(* IEC 61131-3 sources: volt/packages/volt-lsp-iec/test-corpus/pro2193/Device/Plc Logic/Application/09 Misc/Library Manager/L_MC1P_MotionControlBasic, 598 files *)

(* ---- L_MC1P_ABC_STATE.dut ---- *)
TYPE L_MC1P_ABC_STATE :
(
	STANDBY := 0,
	STOP := 1,
	HOMING := 2,
	JOGGING := 3,
	MOVEVEL := 4,
	MOVEABS := 5,
	MOVEREL := 6,
	EXTERNAL := 7,
	ERROR := 8,
	FINISHPOSITIONING := 9
);
END_TYPE

(* ---- L_MC1P_ADDITIONALCONFIGINFO.dut ---- *)
TYPE L_MC1P_ADDITIONALCONFIGINFO :
STRUCT
	LWIDENTDRIVESWITCHOFF : LWORD := 0;
	DWREVISION : DWORD := 0;
	DWMOTORRATEDSPEED : DWORD := 3000;
	LRREFCURRENTMOTOR : LREAL := 0;
	LRREFTORQUEMOTOR : LREAL := 1;
	LRMOTORRATEDTORQUE : LREAL := 1;
	LRTORQUELIMITFACTOR : LREAL := 1;
	LRINERTIAMOTOR : LREAL := 0.01;
	DWMOTORREVOLUTION : DWORD := 1;
	DWENCODERCRC : DWORD := 0;
	XRESETRETAINENCERRORAFTERMAINSWITCH : BOOL;
	XFEEDBACKABSPOSAVAILABLE : BOOL := TRUE;
	XVFCMODE : BOOL := FALSE;
	XTACIA402ADVANCED : BOOL := FALSE;
	WMCTRLMODEDRIVE : USINT := 1;
	XDRIVELOADENCODER : BOOL := FALSE;
	DWDRIVELOADENCODERFEEDBACKCONFIG : DWORD := 0;
	DWDRIVELOADENCODERORIENTATION : DWORD := 0;
	DWDRIVELOADENCODERCRC : DWORD := 0;
	XDEVICETRANSMITTIMESVALID : BOOL;
	LRDEVICETRANSMITTIMEACTPOSMS : LREAL;
	LRDEVICETRANSMITTIMESETPOSMS : LREAL;
END_STRUCT
END_TYPE

(* ---- L_MC1P_ADDITIONALLIMITS.dut ---- *)
TYPE L_MC1P_ADDITIONALLIMITS :
(
	NOTACTIVE := 0,
	ADDITIONALPOSLIMITS := 1
);
END_TYPE

(* ---- L_MC1P_AUTOTUNINGPARA.dut ---- *)
TYPE L_MC1P_AUTOTUNINGPARA :
STRUCT
	MAXVELOCITY : LREAL;
	MAXACCELERATION : LREAL := 0;
	MAXDISTANCE : LREAL := 0;
	MOVEMENTDISTANCE : LREAL := 0;
	STATE : WORD := 0;
	COMMANDIN : USINT;
	VPNFACTOR : WORD;
	TNNFACTOR : WORD;
	VPPFACTOR : WORD;
	VPPFACTOREXT : WORD;
	WAITINGTIME : LREAL;
END_STRUCT
END_TYPE

(* ---- L_MC1P_AXIS_STATE.dut ---- *)
TYPE L_MC1P_AXIS_STATE :
(
	ERRORSTOP := 1,
	DISABLED := 2,
	STANDSTILL := 3,
	STOPPING := 4,
	DISCMOTION := 5,
	SYNCMOTION := 6,
	CONTMOTION := 7,
	HOMING := 8,
	SERVICE := 10
);
END_TYPE

(* ---- L_MC1P_AXISBASICCONTROLINSTANCEDATA.dut ---- *)
TYPE L_MC1P_AXISBASICCONTROLINSTANCEDATA :
STRUCT
	XERROR : BOOL;
	EERRORID : L_IE1P_Error;
	XFUNBUSY : BOOL;
	XFUNDONE : BOOL;
	XFUNCOMMANDABORTED : BOOL;
	EFUNSTATEACT : L_MC1P_ABC_State;
	ABCFUNID : WORD;
	WPOWID : WORD;
	XEXIT : BOOL;
	XMOVEVELEXECUTEOLD : BOOL;
	XMOVEABSEXECUTEOLD : BOOL;
	XMOVERELEXECUTEOLD : BOOL;
	XFINISHPOSITIONINGOLD : BOOL;
	XHOMEEXECUTEOLD : BOOL;
	XJOGGINGNEGOLD : BOOL;
	XJOGGINGPOSOLD : BOOL;
	XSTOPOLD : BOOL;
	XHALTOLD : BOOL;
	XABORTOLD : BOOL;
	XPOWERROROLD : BOOL;
	XDISABLESWLIMITOLD : BOOL;
	XFUNDONEOLD : BOOL;
	XRESETHOMEPOSITIONOLD : BOOL;
	XSAVEMOVEVELDONE : BOOL;
	XACYCLICAXIS : BOOL;
	XQSPAPPLDETECTED : BOOL;
	FBSTOP_EXECUTE : BOOL;
	FBHALT_EXECUTE : BOOL;
	FBABORT_EXECUTE : BOOL;
	FBMOVEABS_EXECUTE : BOOL;
	FBMOVEVEL_EXECUTE : BOOL;
	FBMOVEREL_EXECUTE : BOOL;
	FBFINISHPOSITIONING_XFINISHPOSITIONING : BOOL;
	FBFINISHPOSITIONING_XENABLE : BOOL;
	FBJOG_XJOGPOSITIVE : BOOL;
	FBJOG_XJOGNEGATIVE : BOOL;
	FBHOME_EXECUTE : BOOL;
	FBSTOP_XINUSE : BOOL;
	FBHALT_XINUSE : BOOL;
	FBABORT_XINUSE : BOOL;
	FBMOVEABS_XINUSE : BOOL;
	FBMOVEVEL_XINUSE : BOOL;
	FBMOVEREL_XINUSE : BOOL;
	FBFINISHPOSITIONING_XINUSE : BOOL;
	FBJOG_XINUSE : BOOL;
	FBHOME_XINUSE : BOOL;
	FBBASEOLD : POINTER TO L_MC1P_Template_ForAxis;
	FBSTOP_FBBASESTATUS : L_MC1P_Template_ForAxis;
	FBHALT_FBBASESTATUS : L_MC1P_Template_ForAxis;
	FBABORT_FBBASESTATUS : L_MC1P_Template_ForAxis;
	FBHOME_FBBASESTATUS : L_MC1P_Template_ForAxis;
	FBJOG_FBBASESTATUS : L_MC1P_Template_ForAxis;
	FBMOVEABS_FBBASESTATUS : L_MC1P_Template_ForAxis;
	FBMOVEVEL_FBBASESTATUS : L_MC1P_Template_ForAxis;
	FBMOVEREL_FBBASESTATUS : L_MC1P_Template_ForAxis;
	FBFINISHPOSITIONING_FBBASESTATUS : L_MC1P_Template_ForAxis;
	FBSETFASTSTOP_FBBASESTATUS : L_MC1P_Template_ForAxis;
	FBSETFASTSTOP : L_MC1P_SetFastStop_Internal;
	FBRESET_FBBASESTATUS : L_MC1P_Template_ForAxis;
	FBRESET : L_MC1P_Reset_Internal;
	FBSETOVERRIDE_FBBASESTATUS : L_MC1P_Template_ForAxis;
	FBSETOVERRIDE : L_MC1P_SetOverride_Internal;
	FBREADMOTIONSTATE_FBBASESTATUS : L_MC1P_Template_ForAxis;
	FBREADMOTIONSTATE : L_MC1P_ReadMotionState_Internal;
	FBREADAXISERROR_FBBASESTATUS : L_MC1P_Template_ForAxis;
	FBREADAXISERROR : L_MC1P_ReadAxisError_Internal;
END_STRUCT
END_TYPE

(* ---- L_MC1P_AXISEXTENSIONTYPES.dut ---- *)
TYPE L_MC1P_AXISEXTENSIONTYPES :
(
	EMPTY := 0,
	HL9400_ECAT := 1,
	HL9400_CAN := 2,
	I500_ECAT := 3,
	I500_CAN := 4,
	I700 := 5,
	I750 := 6,
	I950 := 7,
	I950ADV := 8,
	I950_DRIVE := 9,
	I950_DRIVECIA := 10,
	GENERICDRIVE := 11,
	ENCFREE := 101,
	ENCIO_BPB := 102,
	ENCIO_ECAT := 103,
	ENCI900_ECAT := 104,
	ENCI900_DRIVE := 105,
	ENCI900_DRIVECIA := 106,
	ENCI500_ECAT := 107
);
END_TYPE

(* ---- L_MC1P_AXISFUNCTION.dut ---- *)
TYPE L_MC1P_AXISFUNCTION :
(
	SIMPLEMODE := 1,
	PLI := 2,
	MOL := 3,
	POSCTRLADAPT := 4,
	SPEEDCTRLADAPT := 5,
	SPEEDCTRLLOAD := 6,
	BRAKEGRINDIN := 7,
	BRAKETEST := 8,
	BASICBRAKECTRLONLYINDRIVE := 9,
	FLEXIBLEMAPPING := 10,
	ZEROPULS2NDFEEDBACK := 11,
	FDBSTATUSBITSAVAILABLE := 12,
	AUTOTUNING := 13,
	PARSAVEINDRIVE := 14
);
END_TYPE

(* ---- L_MC1P_AXISGUID.dut ---- *)
TYPE L_MC1P_AXISGUID :
STRUCT
	ADWDATA : ARRAY [1..4] OF DWORD;
END_STRUCT
END_TYPE

(* ---- L_MC1P_AXISPROPERTIES.dut ---- *)
TYPE L_MC1P_AXISPROPERTIES :
STRUCT
	XVIRTUAL : BOOL := FALSE;
	XTPSUPPORTED : BOOL := FALSE;
	XTPWITHTIMESTAMP : BOOL := FALSE;
	SNTPMAXCHANNEL : SINT := 0;
	XSUPPORTBRAKE : BOOL := FALSE;
	XSUPPORTDCBRAKE : BOOL := FALSE;
	XCHECKCOMMUNICATIONSTATE : BOOL := TRUE;
	XDRIVEHOMINGSUPPORTED : BOOL := FALSE;
	XTACIAADVANCED : BOOL := FALSE;
	BYDELAYLIMITDRIVEOPERATIONENABLED : BYTE := 2;
	LRTRANSMITCYCLESACTPOS : LREAL;
	LRTRANSMITCYCLESSETPOS : LREAL;
	DWTPDELAYACTPOS : DWORD;
	XFORWARDECATSLAVEERROR : BOOL := FALSE;
	XFORCEACYCLICMODE : BOOL := FALSE;
	WOFFSETDRIVEPARA : WORD := 0;
END_STRUCT
END_TYPE

(* ---- L_MC1P_AXISRETAININFO.dut ---- *)
TYPE L_MC1P_AXISRETAININFO :
STRUCT
	MEMTYPE : BYTE;
	MEMVERSION : BYTE;
	MEMLENGTH : WORD;
END_STRUCT
END_TYPE

(* ---- L_MC1P_AXISRETAININFORMATION.dut ---- *)
TYPE L_MC1P_AXISRETAININFORMATION :
STRUCT
	AXISGUID : L_MC1P_AxisGUID;
	ITFRETAIN : L_MC1P_IRetainFunction;
	PDATA : POINTER TO DWORD;
	PDATAMIRROR : POINTER TO DWORD;
END_STRUCT
END_TYPE

(* ---- L_MC1P_AXISSIMIODATA.dut ---- *)
TYPE L_MC1P_AXISSIMIODATA :
STRUCT
	XSTO : BOOL;
	XDIGIN1 : BOOL;
	XDIGIN2 : BOOL;
	XSTIMULATEERROR : BOOL;
	DWERRORCODE : DWORD;
	XQSPONERROR : BOOL;
	XSTIMULATEWARNING : BOOL;
	DWWARNINGCODE : DWORD;
	ETPMODE : UINT := 0;
	LRTPDISTANCE : LREAL;
	LRTPDISTANCEINTERNAL : LREAL;
END_STRUCT
END_TYPE

(* ---- L_MC1P_AXISSIMULATIONPDODATAFROMDRIVE.dut ---- *)
TYPE L_MC1P_AXISSIMULATIONPDODATAFROMDRIVE :
STRUCT
	UICIASTATUSWORD : UINT;
	UILENZESTATUSWORD : UINT;
	SIMODEOFOPERATIONDISP : SINT;
	UIERRORCODE : UINT;
	UITEXTREFID : UINT;
	DIVELACTVALUE : DINT;
	ITORQUEACTVALUE : INT;
	DIPOSACTVALUE : DINT;
	DIFOLLOWINGERRORACTVALUE : DINT;
	IVLACTUALVEL : INT;
	UITPSTATUS : UINT;
	DITPPOS1POSVALUE : DINT;
	DITPPOS1NEGVALUE : DINT;
	DITPPOS2POSVALUE : DINT;
	DITPPOS2NEGVALUE : DINT;
	UILENZESTATUSWORD2 : UINT;
	UDIDIGITALINPUTS : UDINT;
END_STRUCT
END_TYPE

(* ---- L_MC1P_AXISSIMULATIONPDODATAFROMDRIVESCALED.dut ---- *)
TYPE L_MC1P_AXISSIMULATIONPDODATAFROMDRIVESCALED :
STRUCT
	UICIASTATUSWORD : UINT;
	UILENZESTATUSWORD : UINT;
	SIMODEOFOPERATIONDISP : SINT;
	UIERRORCODE : UINT;
	UITEXTREFID : UINT;
	LRVELACTVALUE : LREAL;
	LRTORQUEACTVALUE : LREAL;
	LRPOSACTVALUE : LREAL;
	LRFOLLOWINGERRORACTVALUE : LREAL;
	UITPSTATUS : UINT;
	LRTPPOS1POSVALUE : LREAL;
	LRTPPOS1NEGVALUE : LREAL;
	LRTPPOS2POSVALUE : LREAL;
	LRTPPOS2NEGVALUE : LREAL;
	UILENZESTATUSWORD2 : UINT;
	UDIDIGITALINPUTS : UDINT;
END_STRUCT
END_TYPE

(* ---- L_MC1P_AXISSIMULATIONPDODATATODRIVE.dut ---- *)
TYPE L_MC1P_AXISSIMULATIONPDODATATODRIVE :
STRUCT
	UICTRLWORD : UINT;
	UILENZECTRLWORD : UINT;
	SIMODEOFOPERATION : SINT;
	ITORQUEOFFSET : INT;
	DITARGETPOSITION : DINT;
	DIVELOCITYOFFSET : DINT;
	ISPDCTRL_ILOADVALUE : INT;
	ITARGETTORQUE : INT;
	DITARGETVELOCITY : DINT;
	IVLTARGETVEL : INT;
	UITPFUNCTION1 : UINT;
	UIPOSTORQUELIMIT : UINT;
	UINEGTORQUELIMIT : UINT;
	DIUPPERSPEEDLIMIT : DINT;
	DILOWERSPEEDLIMIT : DINT;
END_STRUCT
END_TYPE

(* ---- L_MC1P_AXISSIMULATIONPDODATATODRIVESCALED.dut ---- *)
TYPE L_MC1P_AXISSIMULATIONPDODATATODRIVESCALED :
STRUCT
	UICTRLWORD : UINT;
	UILENZECTRLWORD : UINT;
	SIMODEOFOPERATION : SINT;
	LRSETPOSITION : LREAL;
	LRSETVELOCITY : LREAL;
	LRSETTORQUE : LREAL;
	LRSPDCTRL_ILOADVALUE : LREAL;
	LRVLTARGETVELOCITY : LREAL;
	UITPFUNCTION1 : UINT;
	LRPOSTORQUELIMIT : LREAL;
	LRNEGTORQUELIMIT : LREAL;
	LRUPPERSPEEDLIMIT : LREAL;
	LRLOWERSPEEDLIMIT : LREAL;
END_STRUCT
END_TYPE

(* ---- L_MC1P_AXISSIMULATIONSDODATA.dut ---- *)
TYPE L_MC1P_AXISSIMULATIONSDODATA :
STRUCT
	LRRATEDMOTORTORQUE : LREAL := 0.6;
	LRRATEDMOTORSPEED : LREAL := 4050;
	LRINERTIAMOTOR : LREAL := 0.14;
	LRINERTIALOAD : LREAL := 0;
	LRMOTORRATEDCURRENT : LREAL := 1.8;
	LRMAXMOTORSPEED : LREAL := 6075;
	BYMCTRLMODE : BYTE := 1;
	LRVP_SPEEDCTRL : LREAL := 0.00045;
	LRTN_SPEEDCTRL : LREAL := 12.8;
	LRVP_POSCTRL : LREAL := 28.4;
	LRPOSCTRLOUTPUTLIMITATION : LREAL := 480000;
	UIINSABILITYVALUE : UINT;
	UIINSABILITYINDICATOR : USINT;
	USISWITCHINGFREQUENCY : USINT := 1;
	LRPOSCTRLADAPT : LREAL := 100.0;
	LRSPEEDCTRLADAPT : LREAL := 100.0;
	LRMAXTORQUE : LREAL := 250.0;
	LRSPEEDFILTERTIME : LREAL := 0.3;
	WNBRORREVOLUTION : WORD := 1;
	DWINKPERREV : DWORD := 65536;
	DWENCODERCRC : DWORD := 1234;
	DWENCODERCRCLOAD : DWORD := 4567;
	USIBRAKEMODE : USINT := 2;
	UIBRAKESRCOFSTARTINGTORQUE : UINT := 1;
	LRBRAKEDETECTEDSTARTINGTORQUE : LREAL := 0;
	LRBRAKERELEASINGTIME : LREAL := 0.1;
	LRBRAKECLOSINGTIME : LREAL := 0.1;
	USIBRAKEOVERRIDE : USINT := 0;
	LRSTARTTORQUE : LREAL;
	UIBRAKELOGICSTATE : UINT;
	UICONTROLMODECIA402ADVANCED : UINT := 0;
	LRVP_LOADPOSCTRL : LREAL := 20.0;
	SIIPOTIMEEXP : SINT;
	USIIPOTIME : USINT;
	UIQSPOPTION : UINT;
	UDIPOSITIONREACHEDWINDOW : UDINT := 1000;
	UDIQSPDECELERATION : UDINT := 2147483647;
	DWREVISIONNBR : DWORD := 16#20000;
	DWFIRSTSYNCTIME : DWORD;
	USISPEEDERRORRESPONSE : USINT;
	SSWVERSION : STRING(50) := '1.7.5.2420 (release)';
	USIDISABLEPDOS : USINT;
	USIDRIVECOMMAND_0X2825 : USINT;
	UDIMAINSWITCHINGCYCLES_0X2D81_4 : UDINT := 666;
	USIPOSSETMODE_0X2984 : USINT;
	LRVLACCDELTASPEED : LREAL := 0;
	LRVLACCDELTATIME : LREAL := 10;
	LRVLDECDELTASPEED : LREAL := 0;
	LRVLDECDELTATIME : LREAL := 0;
	BYDISABLEDEVICE : BYTE;
	LRADDSPEEDLIMITATION : LREAL := 0;
	AUIGAINCHARACTERISTIC : ARRAY [1..11] OF WORD := [10, 100, 100, 100, 1000, 100, 2000, 100, 5000, 100, 0];
END_STRUCT
END_TYPE

(* ---- L_MC1P_AXISSLOT.dut ---- *)
TYPE L_MC1P_AXISSLOT :
(
	AXISA := 16#0,
	AXISB := 16#800
);
END_TYPE

(* ---- L_MC1P_BACKLASHCONTACTSTATE.dut ---- *)
TYPE L_MC1P_BACKLASHCONTACTSTATE :
(
	NOCONTACT := 0,
	NEGATIVECONTACT := 1,
	POSITIVECONTACT := 2
);
END_TYPE

(* ---- L_MC1P_BRAKEAUTOSTATE.dut ---- *)
TYPE L_MC1P_BRAKEAUTOSTATE :
(
	AS_IDLE,
	AS_RAMPDOWN,
	AS_CLOSINGBRAKE,
	AS_INITBRAKECLOSE,
	AS_BRAKECLOSED,
	AS_RELEASINGBRAKE,
	AS_SUPERVISORMODE,
	AS_DIRECTCONTROL
);
END_TYPE

(* ---- L_MC1P_BRAKECMDBRAKEGRINDINPARA.dut ---- *)
TYPE L_MC1P_BRAKECMDBRAKEGRINDINPARA :
STRUCT
	MOTORSPEED : INT := 1000;
	RAMPTIME : INT := 1000;
	ONTIME : INT := 500;
	OFFTIME : INT := 500;
	CYCLES : WORD := 4;
	GRINDINCONTROL : BYTE;
	MODE : USINT;
	CYCLESOUT : WORD;
	STATE : WORD;
	POSLIMIT1 : LREAL;
	POSLIMIT2 : LREAL;
END_STRUCT
END_TYPE

(* ---- L_MC1P_BRAKECMDBRAKETESTPARA.dut ---- *)
TYPE L_MC1P_BRAKECMDBRAKETESTPARA :
STRUCT
	MOTORTORQUE : DINT := 0;
	RAMPTIME : INT := 1000;
	HOLDTIME : INT := 4000;
	POSTHRESHOLD : INT;
	STATE : WORD := 0;
	WBRAKETESTMODE : USINT;
END_STRUCT
END_TYPE

(* ---- L_MC1P_BRAKECTRL.dut ---- *)
TYPE L_MC1P_BRAKECTRL :
STRUCT
	XDISABLEPHIERR : BOOL;
	XBRAKEFQSP : BOOL;
	XTORQUETIMEOUT : BOOL;
	XRELEASED : BOOL;
	XOUTPUTRELEASEOLD : BOOL;
	XOBSERVE : BOOL;
	XMODULENOTOK : BOOL;
	XEXTSIGNOTOK : BOOL;
	XMODULEFEEDBACK : BOOL;
	XBRAKEOPENED : BOOL;
	XBRAKECLOSED : BOOL;
	XINVERTBRAKE : BOOL;
	XINVERTBRAKEOLD : BOOL;
	XUVDETECTEDOLD : BOOL;
	XACTSPEEDBELOWMINSPEED : BOOL;
	XBIT15 : BOOL;
END_STRUCT
END_TYPE

(* ---- L_MC1P_BRAKEERRORCODES.dut ---- *)
TYPE L_MC1P_BRAKEERRORCODES :
(
	EC_POSITIONDRIFT := 3,
	EC_POSITIONDRIFTCINH := 11,
	EC_RAMPWATCH := 4,
	EC_ERRORMODULE := 5,
	EC_ERROREXTSIGNAL := 13,
	EC_ERRORTORQUETIMEOUT := 18,
	EC_ERRORBRAKESTATEINVALID := 19,
	EC_ERRORBRAKEMODEINVALID := 20,
	EC_TORQUELIMITED := 30
);
END_TYPE

(* ---- L_MC1P_BRAKEGRINDINSTATE.dut ---- *)
TYPE L_MC1P_BRAKEGRINDINSTATE :
(
	NOTACTIVE := 0,
	INIT := 1,
	BRAKEGRINDIN := 3,
	DONE := 4,
	ERROR := 5,
	ABORTED := 6
);
END_TYPE

(* ---- L_MC1P_BRAKELOGICSTATE.dut ---- *)
TYPE L_MC1P_BRAKELOGICSTATE :
(
	OFF := 0,
	WAITON := 1,
	SELECTPRETORQUE := 10,
	LOADPRETORQUE := 11,
	OPENBRAKE := 20,
	OPERATION := 30,
	CLOSEBRAKE := 40,
	TURNOFF := 50
);
END_TYPE

(* ---- L_MC1P_BRAKEMODE.dut ---- *)
TYPE L_MC1P_BRAKEMODE :
(
	OFF := 0,
	MANUALCONTROL_PLC := 1,
	AUTOMATIC_PLC := 2
);
END_TYPE

(* ---- L_MC1P_BRAKEOUTSTATE.dut ---- *)
TYPE L_MC1P_BRAKEOUTSTATE :
STRUCT
	XBRAKECONTROLACTIVE : BOOL;
	XMODULEOPERATION : BOOL;
	XBRAKEOUTSTATE : BOOL;
	XTORQUECTRLACTIVE : BOOL;
	XBRAKECINH : BOOL;
	XERRORACTIVE : BOOL;
	XGRINDINACTIVE : BOOL;
	XTORQUETESTACTIVE : BOOL;
	XMANOPERATION : BOOL;
	XAUTOPERATION : BOOL;
	XERROREXTFEEDBACK : BOOL;
	XERRORPOSDRIFT : BOOL;
	XERRORBRAKEMODULE : BOOL;
	XINFOTIMEOUTACTIVATE : BOOL;
	XGRINDINDONE : BOOL;
	XTORQUETESTDONE : BOOL;
	XERRORTORQUECTRL : BOOL;
	XACTSPEEDBELOWMIN : BOOL;
	XERRORTORQUELIMITED : BOOL;
END_STRUCT
END_TYPE

(* ---- L_MC1P_BRAKEPARA.dut ---- *)
TYPE L_MC1P_BRAKEPARA :
STRUCT
	LRRELEASETIME : LREAL;
	LRACTIVATIONTIME : LREAL;
	DWBRAKEMODE : DWORD;
	ESELBRAKEMODE : DWORD;
	LRSAMPLEDBRAKETORQUE : LREAL;
	LREFFECTIVESTARTINGTORQUE : LREAL;
	ALRMSTARTVALUE : ARRAY [1..2] OF LREAL;
	LRBRAKERAMPTIME : LREAL;
	XBRAKEACCDEPENDING : BOOL;
	WSOURCESTARTVALUE : WORD;
END_STRUCT
END_TYPE

(* ---- L_MC1P_BRAKESTATE.dut ---- *)
TYPE L_MC1P_BRAKESTATE :
(
	EBS_DEFAULT := 0,
	EBS_BRAKECLOSED,
	EBS_BRAKEOPEN,
	EBS_BRAKESWITCHING,
	EBS_BRAKEOBSERVATION,
	EBS_BRAKEAUTO,
	EBS_BRAKEAUTOGSB,
	EBS_BRAKEAUTOSUPERVISOR,
	EBS_BRAKEMANUAL,
	EBS_BRAKEOFF,
	EBS_STATESWITCH,
	EBS_STATEOPERATION
);
END_TYPE

(* ---- L_MC1P_BRAKETESTMODE.dut ---- *)
TYPE L_MC1P_BRAKETESTMODE :
(
	NOLOADTORQUE := 0,
	LOADTORQUEIDENTIFICATION := 1
);
END_TYPE

(* ---- L_MC1P_BRAKETESTSTATE.dut ---- *)
TYPE L_MC1P_BRAKETESTSTATE :
(
	NOTACTIVE := 0,
	INIT := 1,
	TORQUEIDENTIFICATION := 2,
	BRAKETEST := 3,
	DONE := 4,
	ERROR := 5,
	ABORTED := 6
);
END_TYPE

(* ---- L_MC1P_BUFFERDATA.dut ---- *)
TYPE L_MC1P_BUFFERDATA :
STRUCT
	LRBUFFERPOSITIONPOS : LREAL;
	LRBUFFERPOSITIONNEG : LREAL;
	LRBUFFERVELPOS : LREAL;
	LRBUFFERVELNEG : LREAL;
END_STRUCT
END_TYPE

(* ---- L_MC1P_CLASSID.dut ---- *)
TYPE L_MC1P_CLASSID :
(
	AXIS_REF := (L_MC1P_Internal.cdiEnumStartValue + 2),
	AXISBASICCONTROLV2 := (L_MC1P_Internal.cdiEnumStartValue + 3)
);
END_TYPE

(* ---- L_MC1P_COMPENSATIONMODE.dut ---- *)
TYPE L_MC1P_COMPENSATIONMODE :
(
	OFF := 0,
	AUTOMATICSET := 1,
	AUTOMATICACT := 2,
	MANUALLY := 3
);
END_TYPE

(* ---- L_MC1P_CONTROLMODE.dut ---- *)
TYPE L_MC1P_CONTROLMODE :
(
	POSCTRLDRIVE := 0,
	POSCTRLPLC := 1,
	SPEEDCTRLDRIVE := 10,
	TORQUECTRLDRIVE := 20
);
END_TYPE

(* ---- L_MC1P_CONTROLMODESET.dut ---- *)
TYPE L_MC1P_CONTROLMODESET :
(
	POSCTRLDRIVE := 0,
	POSCTRLPLC := 1,
	SPEEDCTRLDRIVE := 10
);
END_TYPE

(* ---- L_MC1P_CTRLABC.dut ---- *)
TYPE L_MC1P_CTRLABC :
STRUCT
	XREGULATORON : BOOL;
	XRESETERROR : BOOL;
	XENABLEPOSITIVE : BOOL := TRUE;
	XENABLENEGATIVE : BOOL := TRUE;
	XDISABLESWLIMIT : BOOL;
	LROVERRIDE : LREAL := 1.0;
	LROVERRIDEACC : LREAL := 1.0;
	LROVERRIDEJERK : LREAL := 1.0;
	XSTOP : BOOL;
	LRSTOPDEC : LREAL := 360000;
	LRSTOPJERK : LREAL := 0;
	XJOGGINGPOS : BOOL;
	XJOGGINGNEG : BOOL;
	XCONTINUOUSUPDATE : BOOL;
	XMOVEVELEXECUTE : BOOL;
	XMOVEABSEXECUTE : BOOL;
	XMOVERELEXECUTE : BOOL;
	XHALT : BOOL;
	LRSETPOS_DIST : LREAL;
	ESETDIRECTION : MC_DIRECTION := MC_DIRECTION.mcPositiveDirection;
	XHOMEEXECUTE : BOOL;
	LRHOMEPOSITION : LREAL;
	XUSEHOMEEXTPARAMETER : BOOL;
	SCHOMEEXTPARAMETER : L_MC1P_HomeParameter;
	SCHOMEEXTTP : MC_TRIGGER_REF;
	XHOMEABSSWITCH : BOOL;
END_STRUCT
END_TYPE

(* ---- L_MC1P_DEVICECLASS.dut ---- *)
TYPE L_MC1P_DEVICECLASS :
(
	VIRTUALAXIS := 0,
	REALAXIS := 1,
	ENCODERAXIS := 2
);
END_TYPE

(* ---- L_MC1P_DIRECTION.dut ---- *)
TYPE L_MC1P_DIRECTION :
(
	BOTH := 0,
	DIRECTIONMASTER := 1
);
END_TYPE

(* ---- L_MC1P_DRIVESPECIFICCONTAINER.dut ---- *)
TYPE L_MC1P_DRIVESPECIFICCONTAINER :
UNION
	PDATA : POINTER TO BYTE;
	BASIC : POINTER TO L_MC1P_DriveSpecific_Basic;
	CIA402 : POINTER TO L_MC1P_DriveSpecific_CiA402;
	I500 : POINTER TO L_MC1P_DriveSpecific_i500;
	I700 : POINTER TO L_MC1P_DriveSpecific_i700;
	I750 : POINTER TO L_MC1P_DriveSpecific_i750;
	I950 : POINTER TO L_MC1P_DriveSpecific_i950;
	I950ADV : POINTER TO L_MC1P_DriveSpecific_i950Adv;
	I950DRIVE : POINTER TO L_MC1P_DriveSpecific_i950_Drive;
	HL9400 : POINTER TO L_MC1P_DriveSpecific_9400HL;
	ENC : POINTER TO L_MC1P_DriveSpecific_Enc;
	ENC_BPB : POINTER TO L_MC1P_DriveSpecific_Enc_Bpb;
	ENC_FREE : POINTER TO L_MC1P_DriveSpecific_Enc_Free;
	ENC_I950 : POINTER TO L_MC1P_DriveSpecific_Enc_i950;
	ENC_I500 : POINTER TO L_MC1P_DriveSpecific_Enc_i500;
	ENC_IOECAT : POINTER TO L_MC1P_DriveSpecific_Enc_IOETC;
END_UNION
END_TYPE

(* ---- L_MC1P_DRIVESTATECOLLECTION.dut ---- *)
TYPE L_MC1P_DRIVESTATECOLLECTION :
STRUCT
	BYDRIVESTATE : BYTE;
	XDRIVETESTMODEACTIVE : BOOL;
	XDRIVEQSPACTIVE : BOOL;
	XDRIVEQSPDONE : BOOL;
	XSTOACTIVE : BOOL;
	XCINHACTIVE : BOOL;
	XVOLTAGEENABLED : BOOL;
	XUSEQSPDRIVEINSTEADOFQSPAPPL : BOOL;
	XPDOINTERFACEDISABLED : BOOL;
	XPLNOTVALID : BOOL;
	XPPIACTIVE : BOOL;
	XMAGNETISATIONFINISHED : BOOL;
	XFAULTACTIVE : BOOL;
	XFAULTREACTIONACTIVE : BOOL;
	XFIRSTERRORCYCLE : BOOL;
	XWARNINGACTIVE : BOOL;
	WTEXTREFID : WORD;
	DWDRIVEERRORID : DWORD;
	XSERVICEMODEHANDLINGINDRIVEACTIVE : BOOL;
	XBRAKESTATUSBIT : BOOL;
	XSBCACTIVE : BOOL;
END_STRUCT
END_TYPE

(* ---- L_MC1P_DRIVETYPE.dut ---- *)
TYPE L_MC1P_DRIVETYPE :
(
	VIRTUAL := 0,
	HL9400 := 1,
	I700 := 2,
	ENCODER := 3,
	GENERICDRIVE := 4,
	I500 := 5,
	I900 := 6,
	I900DRIVE := 7,
	I750 := 8,
	UNIVERSAL := 10
);
END_TYPE

(* ---- L_MC1P_ENCODERTYPE.dut ---- *)
TYPE L_MC1P_ENCODERTYPE :
(
	UNKNOWN := 0,
	FREEENCODER := 1,
	BPBENCODER := 2,
	I500ECAT := 3,
	I900ENCDRIVE := 4,
	I900ECAT := 5,
	ECATENCODER := 6
);
END_TYPE

(* ---- L_MC1P_ERRORINFORMATION.dut ---- *)
TYPE L_MC1P_ERRORINFORMATION :
STRUCT
	EERRORID : L_IE1P_Error;
	XWARNING : BOOL;
	PINSTANCE : DWORD := 0;
	TTIMESTAMP : TIME;
	TRESETTIMESTAMP : TIME;
	DWEXTENDEDERRORINFO : DWORD;
	PSINSTANCENAME : POINTER TO STRING;
END_STRUCT
END_TYPE

(* ---- L_MC1P_EXECUTIONINDEX.dut ---- *)
TYPE L_MC1P_EXECUTIONINDEX :
(
	FIRST := 1,
	SECOND := 2
);
END_TYPE

(* ---- L_MC1P_GISEQUENCE_EXFAN_LIMITS.dut ---- *)
TYPE L_MC1P_GISEQUENCE_EXFAN_LIMITS :
(
	EGI_EXFAN_LIMITS_INIT,
	EGI_EXFAN_LIMITS_FIRSTRAMP,
	EGI_EXFAN_LIMITS_SECONDRAMP,
	EGI_EXFAN_LIMITS_GENERATEPULSE,
	EGI_EXFAN_LIMITS_CHECKDISTANCE,
	EGI_EXFAN_LIMITS_CALCULATEMOVETIME,
	EGI_EXFAN_LIMITS_MOVETOLIMIT
);
END_TYPE

(* ---- L_MC1P_GISEQUENCE_EXFAN_NOLIMITS.dut ---- *)
TYPE L_MC1P_GISEQUENCE_EXFAN_NOLIMITS :
(
	EGI_EXFAN_NOLIMITS_INIT,
	EGI_EXFAN_NOLIMITS_FIRSTRAMP,
	EGI_EXFAN_NOLIMITS_SECONDRAMP,
	EGI_EXFAN_NOLIMITS_GENERATEPULSE,
	EGI_EXFAN_NOLIMITS_CHECKDIRECTION
);
END_TYPE

(* ---- L_MC1P_GISEQUENCE_NOEXFAN_LIMITS.dut ---- *)
TYPE L_MC1P_GISEQUENCE_NOEXFAN_LIMITS :
(
	EGI_NOEXFAN_LIMITS_INIT,
	EGI_NOEXFAN_LIMITS_FIRSTRAMP,
	EGI_NOEXFAN_LIMITS_SECONDRAMP,
	EGI_NOEXFAN_LIMITS_GENERATEPULSE,
	EGI_NOEXFAN_LIMITS_WAITONTIME,
	EGI_NOEXFAN_LIMITS_CHECKDISTANCE,
	EGI_NOEXFAN_LIMITS_CALCULATEMOVETIME,
	EGI_NOEXFAN_LIMITS_MOVETOLIMIT
);
END_TYPE

(* ---- L_MC1P_GISEQUENCE_NOEXFAN_NOLIMITS.dut ---- *)
TYPE L_MC1P_GISEQUENCE_NOEXFAN_NOLIMITS :
(
	EGI_NOEXFAN_NOLIMITS_INIT,
	EGI_NOEXFAN_NOLIMITS_FIRSTRAMP,
	EGI_NOEXFAN_NOLIMITS_GENERATEPULSE,
	EGI_NOEXFAN_NOLIMITS_WAITONTIME,
	EGI_NOEXFAN_NOLIMITS_CHECKDIRECTION
);
END_TYPE

(* ---- L_MC1P_GRINDINMODE.dut ---- *)
TYPE L_MC1P_GRINDINMODE :
(
	CW := 1,
	CCW := 2,
	CWCCW := 3,
	CCWCW := 4
);
END_TYPE

(* ---- L_MC1P_GRINDINSEQUENCE.dut ---- *)
TYPE L_MC1P_GRINDINSEQUENCE :
(
	EGI_DEFAULT := 0,
	EGI_INIT,
	EGI_CONTROLMODE,
	EGI_RAMP1,
	EGI_RAMP2,
	EGI_RAMPDOWN,
	EGI_PULS1,
	EGI_PULS2,
	EGI_DISABLE,
	EGI_CHOOSESTEPSEQUENCE,
	EGI_CALLSTEPSEQUENCE1,
	EGI_CALLSTEPSEQUENCE2,
	EGI_CALLSTEPSEQUENCE3,
	EGI_CALLSTEPSEQUENCE4,
	EGI_CALCULATEDOWNRAMPTYPE,
	EGI_DONE
);
END_TYPE

(* ---- L_MC1P_HOMEMODE.dut ---- *)
TYPE L_MC1P_HOMEMODE :
(
	CWTORQUELIMIT := -2,
	CCWTORQUELIMIT := -1,
	SETPOSITIONDIRECT := 0,
	CCWLIMITSWITCHCWTP := 1,
	CWLIMITSWITCHCCWTP := 2,
	CWRPCCWRNTP := 3,
	CCWRPCWRNTP := 5,
	CCWLIMITSWITCH := 17,
	CWLIMITSWITCH := 18,
	CWRPCCWRN := 19,
	CCWRPCWRN := 21,
	CCWTP := 33,
	CWTP := 34,
	SETPOSITIONINANYSTATE := 97,
	SETOFFSETINANYSTATE := 98,
	RESETHOMEINFO := 99,
	DRIVEBASED := 100
);
END_TYPE

(* ---- L_MC1P_HOMEPARAMETER.dut ---- *)
TYPE L_MC1P_HOMEPARAMETER :
STRUCT
	EHOMEMODE : L_MC1P_HomeMode;
	EHOMESTOPMODE : L_MC1P_HomeStopMode;
	LRTARGETPOSITION : LREAL;
	LRVELOCITY1 : LREAL;
	LRVELOCITY2 : LREAL;
	LRACCELERATION1 : LREAL;
	LRACCELERATION2 : LREAL;
	LRJERK : LREAL;
	RTORQUELIMIT : REAL;
	RTORQUETIME : REAL;
	DWTPCONFIG : L_MC1P_HomeTPMode;
	WDRIVEHOMEMODE : WORD;
	ESTOPMODEDIRECTION : MC_DIRECTION;
	LROFFSETPOSITION : LREAL;
END_STRUCT
END_TYPE

(* ---- L_MC1P_HOMESTOPMODE.dut ---- *)
TYPE L_MC1P_HOMESTOPMODE :
(
	STOPPOSITIONING := 0,
	RELATIVEPOSITIONING := 1,
	ABSOLUTEPOSITIONING := 2
);
END_TYPE

(* ---- L_MC1P_HOMETPMODE.dut ---- *)
TYPE L_MC1P_HOMETPMODE :
(
	EXTERNALSOURCE := 0,
	TP1_POSEDGE := 1,
	TP1_NEGEDGE := 2,
	TP1_ANYEDGE := 3,
	TP1_ZEROPULSE := 4,
	TP1_ZEROPULSE2NDFDB := 5,
	TP2_POSEDGE := 11,
	TP2_NEGEDGE := 12,
	TP2_ANYEDGE := 13,
	TP2_ZEROPULSE := 14,
	TP2_ZEROPULSEFDB2ND := 15,
	TP3_POSEDGE := 21,
	TP3_NEGEDGE := 22,
	TP3_ANYEDGE := 23,
	TP3_ZEROPULSE := 24,
	TP3_ZEROPULSEFDB2ND := 25,
	TP4_POSEDGE := 31,
	TP4_NEGEDGE := 32,
	TP4_ANYEDGE := 33,
	TP4_ZEROPULSE := 34,
	TP5_ZEROPULSEFDB2ND := 35
);
END_TYPE

(* ---- L_MC1P_I900REFOFFSETHANDLING.dut ---- *)
TYPE L_MC1P_I900REFOFFSETHANDLING :
STRUCT
	DWSWITCHCYCLECOUNTER : DWORD;
	DIDRIVEREFOFFSET : DINT;
END_STRUCT
END_TYPE

(* ---- L_MC1P_INTERNALBRAKEMODE.dut ---- *)
TYPE L_MC1P_INTERNALBRAKEMODE :
(
	BM_OFF := 0,
	BM_MANINT := 11,
	BM_AUTINT := 12,
	BM_MANEXT := 1,
	BM_AUTEXT := 2,
	BM_AUTGSB := 22
);
END_TYPE

(* ---- L_MC1P_INTERPOLATIONMODE.dut ---- *)
TYPE L_MC1P_INTERPOLATIONMODE :
(
	LINEAR := 0,
	QUADRATICPOS := 1
);
END_TYPE

(* ---- L_MC1P_INTPROFILEDATA.dut ---- *)
TYPE L_MC1P_INTPROFILEDATA :
STRUCT
	PHASE1 : L_MC1P_ProfilePhaseData;
	PHASE2 : L_MC1P_ProfilePhaseData;
	PHASE3 : L_MC1P_ProfilePhaseData;
	PHASE4 : L_MC1P_ProfilePhaseData;
	PHASE5 : L_MC1P_ProfilePhaseData;
	PHASE6 : L_MC1P_ProfilePhaseData;
	PHASE7 : L_MC1P_ProfilePhaseData;
END_STRUCT
END_TYPE

(* ---- L_MC1P_INTPROFILEDATAACC.dut ---- *)
TYPE L_MC1P_INTPROFILEDATAACC :
STRUCT
	PHASE1 : L_MC1P_ProfilePhaseData;
	PHASE2 : L_MC1P_ProfilePhaseData;
	PHASE3 : L_MC1P_ProfilePhaseData;
END_STRUCT
END_TYPE

(* ---- L_MC1P_KINDOFMOTION.dut ---- *)
TYPE L_MC1P_KINDOFMOTION :
(
	NOTDEFINED := 0,
	TRANSLATORY := 1,
	ROTARY := 2
);
END_TYPE

(* ---- L_MC1P_MAPPEDELEMENT.dut ---- *)
TYPE L_MC1P_MAPPEDELEMENT :
STRUCT
	WPARAMETER : WORD;
	WSIZE : WORD;
	PBADRESS : POINTER TO BYTE;
	PADDITIONALDATA : POINTER TO BYTE;
END_STRUCT
END_TYPE

(* ---- L_MC1P_MAPPEDOBJECTS.dut ---- *)
TYPE L_MC1P_MAPPEDOBJECTS :
STRUCT
	INDEXSUBINDEX : DWORD;
	USISIZE : USINT;
	XUSEDBYAXISREF : BOOL;
	PDATA : POINTER TO BYTE;
END_STRUCT
END_TYPE

(* ---- L_MC1P_MCTRLCONTROL.dut ---- *)
TYPE L_MC1P_MCTRLCONTROL :
(
	MCSTANDARD := 0,
	MCUF := 4,
	MCFTC := 5
);
END_TYPE

(* ---- L_MC1P_MINMAXVALUE.dut ---- *)
TYPE L_MC1P_MINMAXVALUE :
STRUCT
	LRMIN : LREAL := 0;
	LRMAX : LREAL := 0;
END_STRUCT
END_TYPE

(* ---- L_MC1P_MOLSTATE.dut ---- *)
TYPE L_MC1P_MOLSTATE :
(
	IDLE := 0,
	CHECKMOLACTIVATION := 1,
	MOLCYCLIC := 2,
	ERROR := 999
);
END_TYPE

(* ---- L_MC1P_MULTIAXISINFO.dut ---- *)
TYPE L_MC1P_MULTIAXISINFO :
STRUCT
	UIDEVICESLOT : UINT;
	UIOFFSETDRIVEPARA : UINT;
	ITFSLAVEMULTIAXISMODULEHANDLER : L_IMHP_IModuleHandler;
	ITFSLAVEAXISMODULEHANDLER : L_IMHP_IModuleHandler;
END_STRUCT
END_TYPE

(* ---- L_MC1P_ORDINALTYPE.dut ---- *)
TYPE L_MC1P_ORDINALTYPE :
(
	OTNONE := 0,
	OTBOOL := 1,
	OTBYTE := 2,
	OTSINT := 3,
	OTUSINT := 4,
	OTWORD := 5,
	OTINT := 6,
	OTUINT := 7,
	OTDWORD := 8,
	OTDINT := 9,
	OTUDINT := 10,
	OTLWORD := 11,
	OTLINT := 12,
	OTULINT := 13,
	OTREAL := 14,
	OTLREAL := 15
);
END_TYPE

(* ---- L_MC1P_PARACCESS.dut ---- *)
TYPE L_MC1P_PARACCESS :
STRUCT
	AXISNAME : REFERENCE TO STRING;
	DEVICETYPE : REFERENCE TO WORD;
	AXISSTATE : REFERENCE TO WORD;
	AXISSTATUSWORD : REFERENCE TO DWORD;
	ACTIVEERRORID : REFERENCE TO WORD;
	AXISCONTROLWORD : REFERENCE TO WORD;
	AXISCONFIGURATION : REFERENCE TO DWORD;
	ACTPOSITION : REFERENCE TO LREAL;
	ACTVELOCITY : REFERENCE TO LREAL;
	ACTACCELERATION : REFERENCE TO LREAL;
	ACTTORQUE : REFERENCE TO LREAL;
	SETPOSITION : REFERENCE TO LREAL;
	SETVELOCITY : REFERENCE TO LREAL;
	SETACCELERATION : REFERENCE TO LREAL;
	SETTORQUE : REFERENCE TO LREAL;
	KINDOFMOTIONSELECTION : REFERENCE TO WORD;
	ACTIVEUNIT : REFERENCE TO WORD;
	RATIONUMERATORADD : REFERENCE TO DWORD;
	RATIODENOMINATORADD : REFERENCE TO DWORD;
	AXISMODE : REFERENCE TO WORD;
	UDITOTALMEASURINGRANGE : REFERENCE TO UDINT;
	USEASVIRTUAL : REFERENCE TO BOOL;
	TRAVERSINGRANGE : REFERENCE TO WORD;
	CYCLELENGTH : REFERENCE TO LREAL;
	FEEDCONSTANT : REFERENCE TO LREAL;
	RATIONUMERATOR : REFERENCE TO DWORD;
	RATIODENOMINATOR : REFERENCE TO DWORD;
	ORIENTATIONINV : REFERENCE TO BOOL;
	INKPERREV : REFERENCE TO DWORD;
	INERTIALOAD : REFERENCE TO LREAL;
	INERTIAMOTOR : REFERENCE TO LREAL;
	REFTORQUE : REFERENCE TO LREAL;
	DEFAULTVELOCITY : REFERENCE TO LREAL;
	DEFAULTACCELERATION : REFERENCE TO LREAL;
	DEFAULTJERK : REFERENCE TO LREAL;
	MOTORRATEDVELOCITY : REFERENCE TO LREAL;
	MAXVELOCITY : REFERENCE TO LREAL;
	MAXACCELERATION : REFERENCE TO LREAL;
	MAXJERK : REFERENCE TO LREAL;
	DECERRORSTOP : REFERENCE TO LREAL;
	JERKERRORSTOP : REFERENCE TO LREAL;
	ENABLESWLIMIT : REFERENCE TO BOOL;
	SWLIMITPOS : REFERENCE TO LREAL;
	SWLIMITNEG : REFERENCE TO LREAL;
	BEHAVEONSWLIMIT : REFERENCE TO WORD;
	ENABLEFOLLOWINGERROR : REFERENCE TO BOOL;
	MAXFOLLOWINGERRORWARNING : REFERENCE TO LREAL;
	MAXFOLLOWINGERRORERROR : REFERENCE TO LREAL;
	ACTFOLLOWINGERROR : REFERENCE TO LREAL;
	MAXFOLLOWINGERROR : REFERENCE TO LREAL;
	FOLLOWINGERRORREACTION : REFERENCE TO WORD;
	ENCODERINPUTFILTER : REFERENCE TO USINT;
	ENCODERPOSFILTERSTATE : REFERENCE TO WORD;
	ENCODERVELFILTERSTATE : REFERENCE TO WORD;
	BTWFILTERTIME : REFERENCE TO DINT;
	REDPOSQUANT : REFERENCE TO WORD;
	ENCFILTERCYCLES : REFERENCE TO WORD;
	ENCFILTERCYCLESPOS : REFERENCE TO WORD;
	COMPENSATIONMODE : REFERENCE TO WORD;
	SETVALDELAYTIME : REFERENCE TO LREAL;
	ENCODERUPDATETIME : REFERENCE TO DWORD;
	HOMING_MODE : REFERENCE TO INT;
	HOMING_STOPMODE : REFERENCE TO INT;
	HOMING_TARGETPOSITION : REFERENCE TO LREAL;
	HOMING_VELOCITY1 : REFERENCE TO LREAL;
	HOMING_VELOCITY2 : REFERENCE TO LREAL;
	HOMING_ACCELERATION1 : REFERENCE TO LREAL;
	HOMING_ACCELERATION2 : REFERENCE TO LREAL;
	HOMING_JERK : REFERENCE TO LREAL;
	HOMING_TORQUELIMIT : REFERENCE TO REAL;
	HOMING_TORQUETIME : REFERENCE TO REAL;
	HOMING_TPCONFIG : REFERENCE TO DWORD;
	HOMING_RESTOREHOMEPOSITION : REFERENCE TO BOOL;
	HOMING_RESTORETRESHOLD : REFERENCE TO LREAL;
	HOMING_DRIVEHOMEMODE : REFERENCE TO WORD;
	HOMING_HOMEPOSITION : REFERENCE TO LREAL;
	HOMING_POSSETPERMANENTLY : REFERENCE TO USINT;
	HOMIN_OFFSETPOSITION : REFERENCE TO LREAL;
	HOMING_STOPMODEDIRECTION : REFERENCE TO INT;
	CONTROLMODEDEFAULT : REFERENCE TO WORD;
	ACTCONTROLMODE : REFERENCE TO WORD;
	ENCODERNAME : REFERENCE TO STRING;
	POSCTRLGAIN : REFERENCE TO LREAL;
	POSCTRLOUTPUTLIMITATION : REFERENCE TO LREAL;
	POSCTRKOUTPUT : REFERENCE TO LREAL;
	POSCTRLADAPTVALUE : REFERENCE TO UINT;
	POSCTRLADAPTIONFROM0X2985 : REFERENCE TO USINT;
	POSCTRLADAPTACTIVEVALUE : REFERENCE TO UINT;
	SETVALUEMONITORING : REFERENCE TO BOOL;
	TIMELIMITSWITCHON : REFERENCE TO REAL;
	REAKTONMCFBERROR : REFERENCE TO BOOL;
	ENABLELOGENTRY : REFERENCE TO BOOL;
	HWLIMITERRORREACTION : REFERENCE TO USINT;
	SWLIMITERRORREACTION : REFERENCE TO USINT;
	LIMITPROFILEERRORREACTION : REFERENCE TO USINT;
	CINHERRORREACTION : REFERENCE TO USINT;
	LIMITERSTOPREACTION : REFERENCE TO USINT;
	BRAKE_MODE : REFERENCE TO DWORD;
	BRAKE_RELEASETIME : REFERENCE TO LREAL;
	BRAKE_ACTIVATIONTIME : REFERENCE TO LREAL;
	BRAKE_ACTMODE : REFERENCE TO DWORD;
	BRAKE_SAMPLEDTORQUE : REFERENCE TO LREAL;
	BRAKE_EFFECTIVETORQUE : REFERENCE TO LREAL;
	BRAKETEST_STATE : REFERENCE TO WORD;
	BRAKE_SOURCESTARTVALUE : REFERENCE TO WORD;
	BRAKE_MSTARTVALUE : REFERENCE TO LREAL;
	BRAKE_BRAKERAMPTIME : REFERENCE TO LREAL;
	BRAKE_BRAKEACCDEPENDING : REFERENCE TO BOOL;
	BRAKETEST_CMD : REFERENCE TO USINT;
	BRAKETEST_MODE : REFERENCE TO USINT;
	BRAKETEST_TORQUE : REFERENCE TO DINT;
	BRAKETEST_THRESHOLD : REFERENCE TO INT;
	BRAKETEST_RAMPTIME : REFERENCE TO INT;
	BRAKETEST_HOLDTIME : REFERENCE TO INT;
	BRAKETEST_ACTTRESHOLD : REFERENCE TO INT;
	TORQUELIMHIGH : REFERENCE TO INT;
	TORQUELIMLOW : REFERENCE TO INT;
	WINDOWTARGETREACHED : REFERENCE TO LREAL;
	WINDOWTARGETREACHEDTIME : REFERENCE TO LREAL;
	WINDOWSTANDSTILL : REFERENCE TO LREAL;
	OPTIMIZEDPROFILECALCULATIONMODE : REFERENCE TO UINT;
	MODPOSTOLERANCE : REFERENCE TO LREAL;
	RECOVERYWINDOWPOS : REFERENCE TO LREAL;
	RECOVERYWINDOWNEG : REFERENCE TO LREAL;
	SERVICEDIRECTION : REFERENCE TO WORD;
	BRAKEGRINDIN_CMD : REFERENCE TO USINT;
	BRAKEGRINDIN_MODE : REFERENCE TO USINT;
	BRAKEGRINDIN_CTRL : REFERENCE TO BYTE;
	BRAKEGRINDIN_SPEED : REFERENCE TO INT;
	BRAKEGRINDIN_RAMPTIME : REFERENCE TO INT;
	BRAKEGRINDIN_ONTIME : REFERENCE TO INT;
	BRAKEGRINDIN_OFFTIME : REFERENCE TO INT;
	BRAKEGRINDIN_CYCLES : REFERENCE TO WORD;
	BRAKEGRINDIN_CYCLESOUT : REFERENCE TO WORD;
	BRAKEGRINDIN_STATE : REFERENCE TO WORD;
	LIMITEDVELOCITY1 : REFERENCE TO LREAL;
	LIMITEDDECELERATION1 : REFERENCE TO LREAL;
	LIMITEDVELOCITY2 : REFERENCE TO LREAL;
	LIMITEDDECELERATION2 : REFERENCE TO LREAL;
	LIMITEDVELOCITY3 : REFERENCE TO LREAL;
	LIMITEDDECELERATION3 : REFERENCE TO LREAL;
	LIMITEDVELOCITY4 : REFERENCE TO LREAL;
	LIMITEDDECELERATION4 : REFERENCE TO LREAL;
	LIMITEDDISTANCE : REFERENCE TO LREAL;
	SLSOFFSETVELOCITY : REFERENCE TO LREAL;
	FOLLOWERSLS : REFERENCE TO BOOL;
	LIMITSPEEDCTRLSLS : REFERENCE TO BOOL;
	DISABLESAFETYINTERFACE : REFERENCE TO DWORD;
	REQUESTSAFETYINTERFACE : REFERENCE TO DWORD;
	SLIDISTANCE : REFERENCE TO LREAL;
	BRAKEGRINDIN_POSLIMIT1 : REFERENCE TO LREAL;
	BRAKEGRINDIN_POSLIMIT2 : REFERENCE TO LREAL;
	AUTOTUNING_CMD : REFERENCE TO USINT;
	AT_VELOCITY : REFERENCE TO LREAL;
	AT_ACCELERATION : REFERENCE TO LREAL;
	AT_DISTANCE : REFERENCE TO LREAL;
	AT_CALCULATEDDISTANCE : REFERENCE TO LREAL;
	AT_VPNFACTOR : REFERENCE TO WORD;
	AT_TNNFACTOR : REFERENCE TO WORD;
	AT_STATE : REFERENCE TO WORD;
	AT_VPPFACTOR : REFERENCE TO WORD;
	AT_VPPFACTOREXT : REFERENCE TO WORD;
	AT_WAITINGTIME : REFERENCE TO LREAL;
	JOGGINGSETVEL : REFERENCE TO LREAL;
	JOGGINGSETACC : REFERENCE TO LREAL;
	JOGGINGSETDEC : REFERENCE TO LREAL;
	JOGGINGSETJERK : REFERENCE TO LREAL;
	HALTDEC : REFERENCE TO LREAL;
	HALTJERK : REFERENCE TO LREAL;
END_STRUCT
END_TYPE

(* ---- L_MC1P_PARAMETERDATASIM.dut ---- *)
TYPE L_MC1P_PARAMETERDATASIM :
STRUCT
	WINDEX : WORD;
	BYSUBINDEX : BYTE;
	PVALUE : POINTER TO BYTE;
	BYNROFBYTE : BYTE;
	XSUPPORTED : BOOL;
	XWRITEACCESS : BOOL;
	XAXISOFFSETSUPPORTED : BOOL;
	EFIXTOLREAL : L_MC1P_ScaleFixToLREAL := L_MC1P_ScaleFixToLREAL.None;
END_STRUCT
END_TYPE

(* ---- L_MC1P_PARAMS.dut ---- *)
TYPE L_MC1P_PARAMS :
(
	AXISNAME := 2,
	DEVICETYPE := 3,
	AXISSTATE := 4,
	AXISSTATUSWORD := 5,
	ACTIVEERRORID := 6,
	AXISCONTROLWORD := 8,
	AXISCONFIGURATION := 9,
	ACTPOSITION := 10,
	ACTVELOCITY := 11,
	ACTACCELERATION := 12,
	ACTTORQUE := 13,
	SETPOSITION := 14,
	SETVELOCITY := 15,
	SETACCELERATION := 16,
	SETTORQUE := 17,
	KINDOFMOTIONSELECTION := 20,
	ACTIVEUNIT := 21,
	RATIONUMERATORADD := 25,
	RATIODENOMINATORADD := 26,
	AXISMODE := 27,
	UDITOTALMEASURINGRANGE := 28,
	USEASVIRTUAL := 29,
	TRAVERSINGRANGE := 30,
	CYCLELENGTH := 31,
	FEEDCONSTANT := 32,
	RATIONUMERATOR := 33,
	RATIODENOMINATOR := 34,
	ORIENTATIONINV := 35,
	INKPERREV := 36,
	INERTIALOAD := 37,
	INERTIAMOTOR := 38,
	REFTORQUE := 39,
	DEFAULTVELOCITY := 40,
	DEFAULTACCELERATION := 41,
	DEFAULTJERK := 43,
	MOTORRATEDVELOCITY := 44,
	MAXVELOCITY := 45,
	MAXACCELERATION := 46,
	MAXJERK := 47,
	DECERRORSTOP := 48,
	JERKERRORSTOP := 49,
	ENABLESWLIMIT := 50,
	SWLIMITPOS := 51,
	SWLIMITNEG := 52,
	BEHAVEONSWLIMIT := 53,
	ENABLEFOLLOWINGERROR := 54,
	MAXFOLLOWINGERRORWARNING := 55,
	MAXFOLLOWINGERRORERROR := 56,
	ACTFOLLOWINGERROR := 57,
	MAXFOLLOWINGERROR := 58,
	FOLLOWINGERRORREACTION := 59,
	ENCODERINPUTFILTER := 60,
	ENCODERPOSFILTERSTATE := 61,
	ENCODERVELFILTERSTATE := 62,
	BTWFILTERTIME := 63,
	REDPOSQUANT := 64,
	ENCFILTERCYCLES := 65,
	ENCFILTERCYCLESPOS := 66,
	COMPENSATIONMODE := 67,
	SETVALDELAYTIME := 68,
	ENCODERUPDATETIME := 69,
	HOMING_MODE := 70,
	HOMING_STOPMODE := 71,
	HOMING_TARGETPOSITION := 72,
	HOMING_VELOCITY1 := 73,
	HOMING_VELOCITY2 := 74,
	HOMING_ACCELERATION1 := 75,
	HOMING_ACCELERATION2 := 76,
	HOMING_JERK := 77,
	HOMING_TORQUELIMIT := 78,
	HOMING_TORQUETIME := 79,
	HOMING_TPCONFIG := 80,
	HOMING_RESTOREHOMEPOSITION := 81,
	HOMING_RESTORETRESHOLD := 82,
	HOMING_DRIVEHOMEMODE := 83,
	HOMING_HOMEPOSITION := 84,
	HOMING_POSSETPERMANENTLY := 85,
	HOMIN_OFFSETPOSITION := 86,
	HOMING_STOPMODEDIRECTION := 87,
	CONTROLMODEDEFAULT := 90,
	ACTCONTROLMODE := 91,
	ENCODERNAME := 92,
	POSCTRLGAIN := 93,
	POSCTRLOUTPUTLIMITATION := 94,
	POSCTRKOUTPUT := 95,
	POSCTRLADAPTVALUE := 96,
	POSCTRLADAPTIONFROM0X2985 := 97,
	POSCTRLADAPTACTIVEVALUE := 98,
	SETVALUEMONITORING := 100,
	TIMELIMITSWITCHON := 101,
	REAKTONMCFBERROR := 102,
	ENABLELOGENTRY := 103,
	HWLIMITERRORREACTION := 104,
	SWLIMITERRORREACTION := 105,
	LIMITPROFILEERRORREACTION := 106,
	CINHERRORREACTION := 107,
	LIMITERSTOPREACTION := 108,
	BRAKE_MODE := 110,
	BRAKE_RELEASETIME := 111,
	BRAKE_ACTIVATIONTIME := 112,
	BRAKE_ACTMODE := 113,
	BRAKE_SAMPLEDTORQUE := 114,
	BRAKE_EFFECTIVETORQUE := 115,
	BRAKETEST_STATE := 116,
	BRAKE_SOURCESTARTVALUE := 117,
	BRAKE_MSTARTVALUE := 118,
	BRAKE_BRAKERAMPTIME := 119,
	BRAKE_BRAKEACCDEPENDING := 120,
	BRAKETEST_CMD := 121,
	BRAKETEST_MODE := 122,
	BRAKETEST_TORQUE := 123,
	BRAKETEST_THRESHOLD := 124,
	BRAKETEST_RAMPTIME := 125,
	BRAKETEST_HOLDTIME := 126,
	BRAKETEST_ACTTRESHOLD := 127,
	TORQUELIMHIGH := 128,
	TORQUELIMLOW := 129,
	WINDOWTARGETREACHED := 130,
	WINDOWTARGETREACHEDTIME := 131,
	WINDOWSTANDSTILL := 132,
	OPTIMIZEDPROFILECALCULATIONMODE := 134,
	MODPOSTOLERANCE := 135,
	RECOVERYWINDOWPOS := 136,
	RECOVERYWINDOWNEG := 137,
	SERVICEDIRECTION := 139,
	BRAKEGRINDIN_CMD := 140,
	BRAKEGRINDIN_MODE := 141,
	BRAKEGRINDIN_CTRL := 142,
	BRAKEGRINDIN_SPEED := 143,
	BRAKEGRINDIN_RAMPTIME := 144,
	BRAKEGRINDIN_ONTIME := 145,
	BRAKEGRINDIN_OFFTIME := 146,
	BRAKEGRINDIN_CYCLES := 147,
	BRAKEGRINDIN_CYCLESOUT := 148,
	BRAKEGRINDIN_STATE := 149,
	LIMITEDVELOCITY1 := 150,
	LIMITEDDECELERATION1 := 151,
	LIMITEDVELOCITY2 := 152,
	LIMITEDDECELERATION2 := 153,
	LIMITEDVELOCITY3 := 154,
	LIMITEDDECELERATION3 := 155,
	LIMITEDVELOCITY4 := 156,
	LIMITEDDECELERATION4 := 157,
	LIMITEDDISTANCE := 158,
	SLSOFFSETVELOCITY := 159,
	FOLLOWERSLS := 160,
	LIMITSPEEDCTRLSLS := 161,
	DISABLESAFETYINTERFACE := 162,
	REQUESTSAFETYINTERFACE := 163,
	SLIDISTANCE := 164,
	BRAKEGRINDIN_POSLIMIT1 := 168,
	BRAKEGRINDIN_POSLIMIT2 := 169,
	AUTOTUNING_CMD := 170,
	AT_VELOCITY := 171,
	AT_ACCELERATION := 172,
	AT_DISTANCE := 173,
	AT_CALCULATEDDISTANCE := 174,
	AT_VPNFACTOR := 175,
	AT_TNNFACTOR := 176,
	AT_STATE := 177,
	AT_VPPFACTOR := 178,
	AT_VPPFACTOREXT := 179,
	AT_WAITINGTIME := 180,
	JOGGINGSETVEL := 181,
	JOGGINGSETACC := 182,
	JOGGINGSETDEC := 183,
	JOGGINGSETJERK := 184,
	HALTDEC := 186,
	HALTJERK := 187
);
END_TYPE

(* ---- L_MC1P_PARGENERALMECHANIC.dut ---- *)
TYPE L_MC1P_PARGENERALMECHANIC :
STRUCT
	WBRAKEAVAILABLE : WORD := 0;
	LRBRAKEACTIVATIONTIME : LREAL := 0.01;
	LRCURRCTRLPT2TT_T1 : LREAL := (246.06 * 1E-06);
	LRCURRCTRLPT2TT_T2 : LREAL := (210.35 * 1E-06);
	LRCURRCTRLPT2TT_DELAY : LREAL := (103.3 * 1E-06);
END_STRUCT
END_TYPE

(* ---- L_MC1P_PARMECHANIC.dut ---- *)
TYPE L_MC1P_PARMECHANIC :
STRUCT
	LRINERTIA : LREAL := 2.99E-05;
	LRVISCOSEFACTOR : LREAL := 0.001;
	LRCOULOMBFACTOR : LREAL := 0.025;
	LRCOULOMBSLOPE : LREAL := 1;
	LREXTERNALTORQUE : LREAL;
	LRBRAKEMAXTORQUE : LREAL := 2;
	LRMECHMINPOS : LREAL := 0;
	LRMECHMAXPOS : LREAL := 0;
END_STRUCT
END_TYPE

(* ---- L_MC1P_PARMECHANIC2MS.dut ---- *)
TYPE L_MC1P_PARMECHANIC2MS :
STRUCT
	LRINERTIA2 : LREAL;
	LRD : LREAL;
	LRC : LREAL;
	LRFRICTIONRATIO : LREAL := (1.0 / 4.0);
END_STRUCT
END_TYPE

(* ---- L_MC1P_PARMECHANIC2MS_BACKLASH.dut ---- *)
TYPE L_MC1P_PARMECHANIC2MS_BACKLASH :
STRUCT
	LRBACKLASH : LREAL;
END_STRUCT
END_TYPE

(* ---- L_MC1P_PARMECHANIC3MS.dut ---- *)
TYPE L_MC1P_PARMECHANIC3MS :
STRUCT
	LRINERTIA2 : LREAL := (1.95 - 4);
	LRINERTIA3 : LREAL := 1.6E-05;
	D1 : LREAL := 2.24;
	D2 : LREAL := 0.007;
	C1 : LREAL := 2.24;
	C2 : LREAL := 0.008;
END_STRUCT
END_TYPE

(* ---- L_MC1P_PGFUTVAL.dut ---- *)
TYPE L_MC1P_PGFUTVAL :
STRUCT
	DROUTACC : LREAL;
	DROUTSPEED : LREAL;
	DROUTPOS : LREAL;
	DRCNT : LREAL;
END_STRUCT
END_TYPE

(* ---- L_MC1P_PGPHASENPARA.dut ---- *)
TYPE L_MC1P_PGPHASENPARA :
STRUCT
	DRRELTIME : LREAL;
	DRTIME : LREAL;
	DRRELPOS : LREAL;
	DRPOS : LREAL;
	DRRELSPEED : LREAL;
	DRSPEED : LREAL;
	DRRELACC : LREAL;
	DRACC : LREAL;
	DRJERKA : LREAL;
	IBPROFILENUMBER : INT;
END_STRUCT
END_TYPE

(* ---- L_MC1P_POSCTRLADAPTMODE.dut ---- *)
TYPE L_MC1P_POSCTRLADAPTMODE :
(
	MOTORANDLOAD := 0,
	MOTOR := 1,
	LOAD := 2
);
END_TYPE

(* ---- L_MC1P_POSLINT.dut ---- *)
TYPE L_MC1P_POSLINT :
UNION
	LIPOS : LINT;
	ADIPOS : ARRAY [1..2] OF DINT;
END_UNION
END_TYPE

(* ---- L_MC1P_PPISTATE.dut ---- *)
TYPE L_MC1P_PPISTATE :
(
	IDLE := 0,
	CHECKPPIACTIVATION := 1,
	PPIMONITORING := 2,
	DONE := 3,
	RESETPPIINFORMATION := 4,
	SETPPIINFORMATION := 5,
	ERROR := 999
);
END_TYPE

(* ---- L_MC1P_PRECONTROLMODE.dut ---- *)
TYPE L_MC1P_PRECONTROLMODE :
(
	AUTOMATIC := 0,
	ADDITIVEOFFSETTORQUE := 1,
	EXCLUSIVEOFFSETTORQUE := 2
);
END_TYPE

(* ---- L_MC1P_PRMDATAHEADER.dut ---- *)
TYPE L_MC1P_PRMDATAHEADER :
STRUCT
	PARAMHEADERTYPE : DWORD;
	PARAMETERDATAOFFSETFROMSTARTOF : DWORD;
	PARAMDATASIZE : DWORD;
END_STRUCT
END_TYPE

(* ---- L_MC1P_PRMFILEHEADER.dut ---- *)
TYPE L_MC1P_PRMFILEHEADER :
STRUCT
	PARSETTYPE : DWORD;
	FILEVERSION : DWORD;
	SIZETOTAL : DWORD;
	VENDOR : DWORD;
	PRODUCTCODE : DWORD;
	REVISION : DWORD;
	DATAOFFSET : DWORD;
	DATASIZE : DWORD;
	CRCCHECKSUM : DWORD;
END_STRUCT
END_TYPE

(* ---- L_MC1P_PRMPARAMETERHEADER.dut ---- *)
TYPE L_MC1P_PRMPARAMETERHEADER :
STRUCT
	SIZE : WORD;
	INDEX : WORD;
	SUBINDEX : WORD;
END_STRUCT
END_TYPE

(* ---- L_MC1P_PROFILEDATA.dut ---- *)
TYPE L_MC1P_PROFILEDATA :
STRUCT
	ALRPROFILETIME : ARRAY [0..8] OF LREAL;
	ALRPROFILEPOS : ARRAY [0..8] OF LREAL;
	ALRPROFILEVEL : ARRAY [0..8] OF LREAL;
	ALRPROFILEACC : ARRAY [0..8] OF LREAL;
	ALRPROFILEJERK : ARRAY [0..8] OF LREAL;
END_STRUCT
END_TYPE

(* ---- L_MC1P_PROFILEDATAEXTENDED.dut ---- *)
TYPE L_MC1P_PROFILEDATAEXTENDED :
STRUCT
	ALRPROFILETIME : ARRAY [0..11] OF LREAL;
	ALRPROFILEPOS : ARRAY [0..11] OF LREAL;
	ALRPROFILEVEL : ARRAY [0..11] OF LREAL;
	ALRPROFILEACC : ARRAY [0..11] OF LREAL;
	ALRPROFILEJERK : ARRAY [0..11] OF LREAL;
END_STRUCT
END_TYPE

(* ---- L_MC1P_PROFILEPARAMETER.dut ---- *)
TYPE L_MC1P_PROFILEPARAMETER :
STRUCT
	LRTARGETPOS : LREAL := 0;
	LRTARGETVEL : LREAL := 0;
	LRTARGETACC : LREAL := 0;
	LRMAXVEL : LREAL := 0;
	LRMAXACC : LREAL := 0;
	LRMAXDEC : LREAL := 0;
	LRJERKACC : LREAL := 0;
	LRJERKDEC : LREAL := 0;
END_STRUCT
END_TYPE

(* ---- L_MC1P_PROFILEPHASEDATA.dut ---- *)
TYPE L_MC1P_PROFILEPHASEDATA :
STRUCT
	T : LREAL;
	DS : LREAL;
	DV : LREAL;
	DA : LREAL;
	J : LREAL;
END_STRUCT
END_TYPE

(* ---- L_MC1P_PROFILETYPE.dut ---- *)
TYPE L_MC1P_PROFILETYPE :
(
	POLY_4TH_ORDER := 0,
	POLY_2TH_ORDER := 1,
	POLY_5TH_ORDER := 2
);
END_TYPE

(* ---- L_MC1P_QUICKSTOPOPTION.dut ---- *)
TYPE L_MC1P_QUICKSTOPOPTION :
(
	DISABLEDRIVE := 2,
	STAYINQSP := 6
);
END_TYPE

(* ---- L_MC1P_RETAINDATAENCAXIS.dut ---- *)
TYPE L_MC1P_RETAINDATAENCAXIS :
STRUCT
	XRETAININITIALIZED : BOOL;
	RETAINSTACK1 : L_MC1P_uRetainData;
	RETAINSTACK2 : L_MC1P_uRetainData;
END_STRUCT
END_TYPE

(* ---- L_MC1P_RETAINDATAI700.dut ---- *)
TYPE L_MC1P_RETAINDATAI700 :
STRUCT
	DWENCODERCRC : DWORD;
	LRBRAKESAMPLEDTORQUE : LREAL;
END_STRUCT
END_TYPE

(* ---- L_MC1P_RETAINDATAI700_V2.dut ---- *)
TYPE L_MC1P_RETAINDATAI700_V2 :
STRUCT
	DWENCODERCRC : DWORD;
	LRBRAKESAMPLEDTORQUE : LREAL;
END_STRUCT
END_TYPE

(* ---- L_MC1P_RETAINDATAI700_V3.dut ---- *)
TYPE L_MC1P_RETAINDATAI700_V3 :
STRUCT
	DWENCODERCRC : DWORD;
	LRBRAKESAMPLEDTORQUE : LREAL;
END_STRUCT
END_TYPE

(* ---- L_MC1P_RETAINDATAREALDRIVE.dut ---- *)
TYPE L_MC1P_RETAINDATAREALDRIVE :
STRUCT
	DWPROPERTIES : DWORD;
	UPOSACT : L_MC1P_PosLINT;
	DIREFOFFSETINC : DINT;
	LRACTPOS : LREAL;
	LRABSREFOFFSET : LREAL;
	LRCYCLELENGTH : LREAL;
	LRSCALEFACTOR : LREAL;
END_STRUCT
END_TYPE

(* ---- L_MC1P_RETAINDATAREALDRIVE_V2.dut ---- *)
TYPE L_MC1P_RETAINDATAREALDRIVE_V2 :
STRUCT
	DWPROPERTIES : DWORD;
	UPOSACT : L_MC1P_PosLINT;
	DIREFOFFSETINC : DINT;
	LRACTPOS : LREAL;
	LRABSREFOFFSET : LREAL;
	LRCYCLELENGTH : LREAL;
	LRSCALEFACTOR : LREAL;
	DISETPOSROUNDSLAST : DINT;
	LRLASTSETPOSITION : LREAL;
	DITARGETPOSROUNDS : DINT;
	LRLASTTARGETPOSITION : LREAL;
END_STRUCT
END_TYPE

(* ---- L_MC1P_RETAINDATAREALDRIVE_V3.dut ---- *)
TYPE L_MC1P_RETAINDATAREALDRIVE_V3 :
STRUCT
	DWPROPERTIES : DWORD;
	DIREFOFFSETINC : DINT;
	UPOSACT : L_MC1P_PosLINT;
	LRACTPOS : LREAL;
	LRABSREFOFFSET : LREAL;
	LRCYCLELENGTH : LREAL;
	LRSCALEFACTOR : LREAL;
	LRLASTSETPOSITION : LREAL;
	DISETPOSROUNDSLAST : DINT;
	DITARGETPOSROUNDS : DINT;
	LRLASTTARGETPOSITION : LREAL;
	DRIVEGUID : L_MC1P_AxisGUID;
END_STRUCT
END_TYPE

(* ---- L_MC1P_RETAINDATATYPE.dut ---- *)
TYPE L_MC1P_RETAINDATATYPE :
(
	NONE := -1,
	DATAREALDRIVE := 0,
	DATAI700 := 1
);
END_TYPE

(* ---- L_MC1P_SCALEFIXTOLREAL.dut ---- *)
TYPE L_MC1P_SCALEFIXTOLREAL :
(
	NONE := 0,
	FIX_X := 1,
	FIX_X_X := 10,
	FIX_X_XX := 100,
	FIX_X_XXX := 1000,
	FIX_X_XXXX := 10000,
	FIX_X_XXXXX := 100000
);
END_TYPE

(* ---- L_MC1P_SERVICEDIRECTION.dut ---- *)
TYPE L_MC1P_SERVICEDIRECTION :
(
	BOTH := 0,
	POSITIVE := 1,
	NEGATIVE := 2
);
END_TYPE

(* ---- L_MC1P_SETVALUEMODE.dut ---- *)
TYPE L_MC1P_SETVALUEMODE :
(
	POS := 1,
	VEL := 2,
	POSVEL := 3,
	VELACC := 6,
	POSVELACC := 7,
	VEL_VELFROMPROFILEGEN := 8,
	VEL_VELFROMDIFFPOS := 9
);
END_TYPE

(* ---- L_MC1P_SIMAXISCYCLETIME.dut ---- *)
TYPE L_MC1P_SIMAXISCYCLETIME :
(
	TASKCYCLE_1KHZ := 1,
	TASKCYCLE_2KHZ := 2,
	TASKCYCLE_4KHZ := 4,
	TASKCYCLE_8KHZ := 8,
	TASKCYCLE_16KHZ := 16,
	TASKCYCLE_32KHZ := 32,
	TASKCYCLE_64KHZ := 64
);
END_TYPE

(* ---- L_MC1P_STATUSABC.dut ---- *)
TYPE L_MC1P_STATUSABC :
STRUCT
	XINTERNALCONTROLACTIVE : BOOL;
	XERROR : BOOL;
	EERRORID : L_IE1P_Error;
	XFUNBUSY : BOOL;
	XFUNDONE : BOOL;
	XFUNCOMMANDABORTED : BOOL;
	EFUNSTATEACT : L_MC1P_ABC_State;
	ECONTROLMODE : L_MC1P_ControlMode;
	XISHOMED : BOOL;
	XHWLIMITSWITCHNEG : BOOL;
	XHWLIMITSWITCHPOS : BOOL;
	XSWLIMITENABLED : BOOL;
	XSWLIMITSWITCHNEG : BOOL;
	XSWLIMITSWITCHPOS : BOOL;
	EAXISTYPE : L_MC1P_DriveType;
	EAXISSTATE : L_MC1P_AXIS_STATE;
	XAXISREADY : BOOL;
	XAXISENABLED : BOOL;
	XAXISWARNING : BOOL;
	XAXISERROR : BOOL;
	EAXISERRORID : L_IE1P_Error;
	XDRIVEWARNING : BOOL;
	XDRIVEERROR : BOOL;
	DWDRIVEERRORID : DWORD;
	LRACTPOS : LREAL;
	LRACTVEL : LREAL;
	LRSETPOSOUT : LREAL;
	LRSETVELOUT : LREAL;
	LRACTFOLLOWINGERROR : LREAL;
	XCONSTANTVELOCITY : BOOL;
	XACCELERATING : BOOL;
	XDECELERATING : BOOL;
	XDIRECTIONPOSITIVE : BOOL;
	XDIRECTIONNEGATIVE : BOOL;
	XINPOSITION : BOOL;
	XAXISAVAILABLE : BOOL;
	XSTANDSTILLSETVELOCITY : BOOL;
	XSTANDSTILLACTVELOCITY : BOOL;
	XAXISREADYTOSWITCHON : BOOL;
	XAXISREADYFORMOTION : BOOL;
END_STRUCT
END_TYPE

(* ---- L_MC1P_STOPOPERATION.dut ---- *)
TYPE L_MC1P_STOPOPERATION :
STRUCT
	XSETQSP : BOOL;
	XSETQSPCINH : BOOL;
	XSETCINH : BOOL;
	XSETFASTSTOP : BOOL;
END_STRUCT
END_TYPE

(* ---- L_MC1P_TIMESTAMP.dut ---- *)
TYPE L_MC1P_TIMESTAMP :
STRUCT
	TIME_01 : SysTime;
	TIME_02 : SysTime;
	TIME_03 : SysTime;
	TIME_04 : SysTime;
	TIME_05 : SysTime;
	TIME_06 : SysTime;
	TIME_07 : SysTime;
	TIME_08 : SysTime;
	TIME_DELTA_01_02 : SysTime;
	TIME_DELTA_02_03 : SysTime;
	TIME_DELTA_03_04 : SysTime;
	TIME_DELTA_04_05 : SysTime;
	TIME_DELTA_05_06 : SysTime;
	TIME_DELTA_06_07 : SysTime;
	TIME_DELTA_07_08 : SysTime;
END_STRUCT
END_TYPE

(* ---- L_MC1P_TORQUETESTMONITORING.dut ---- *)
TYPE L_MC1P_TORQUETESTMONITORING :
STRUCT
	PT1_ACTMOTORTORQUE : L_USPP_PT1Filter;
	PT1_SETTORQUE : L_USPP_PT1Filter;
	LRPT1DELAY : LREAL := 0.01;
	ALRSETTORQUE : ARRAY [0..15] OF LREAL;
	LRTORQUETOLERANCE : LREAL := 0.1;
	IDX : UINT;
	XBUFFER : BOOL;
END_STRUCT
END_TYPE

(* ---- L_MC1P_TORQUETESTSEQUENCE.dut ---- *)
TYPE L_MC1P_TORQUETESTSEQUENCE :
(
	ETT_DEFAULT := 0,
	ETT_PREINIT := 9,
	ETT_INIT := 1,
	ETT_CONTROLMODE := 2,
	ETT_TORQUERAMPUP := 3,
	ETT_TORQUERAMPDOWN := 4,
	ETT_CONSTANTWAIT := 5,
	ETT_WAITCINHRELEASE := 6,
	ETT_WAITCINH := 7,
	ETT_IDENTIFYTORQUE := 8,
	ETT_DONE := 10
);
END_TYPE

(* ---- L_MC1P_TPDATA.dut ---- *)
TYPE L_MC1P_TPDATA :
STRUCT
	XSTARTCAPTURING : BOOL;
	XINEXCECUTION : BOOL;
	XNEWEXECUTE : BOOL;
	XCOMMANDABORTED : BOOL;
	NERRORID : INT := 0;
	XVALUESTORED_POSEDGE : BOOL;
	DNRECORDEDPOSITION_POSEDGE : DINT;
	DWTIMESTAMP_POSEDGE : DWORD;
	XNEWVALUESTORED_POSEDGE : BOOL;
	XVALUESTORED_NEGEDGE : BOOL;
	DNRECORDEDPOSITION_NEGEDGE : DINT;
	DWTIMESTAMP_NEGEDGE : DWORD;
	XNEWVALUESTORED_NEGEDGE : BOOL;
	XACTIVATIONLEVEL : BOOL;
	XOVERRIDEACTIVE : BOOL;
	XTIMESTAMPAVAILABLEPOSEDGE : BOOL;
	XTIMESTAMPAVAILABLENEGEDGE : BOOL;
	XPOSITIONAVAILABLEPOSEDGE : BOOL;
	XPOSITIONAVAILABLENEGEDGE : BOOL;
	XACTIVATIONLEVELVALID : BOOL;
END_STRUCT
END_TYPE

(* ---- L_MC1P_TPRECEIVEDATA.dut ---- *)
TYPE L_MC1P_TPRECEIVEDATA :
STRUCT
	XVALUESTORED : BOOL;
	LRRECPOSITION : LREAL;
	DWRECTIMESTAMP : DWORD;
	DWACTTIMESTAMP : DWORD;
	XSUPPORTTIMESTAMP : BOOL;
	XSUPPORTPOSITION : BOOL;
END_STRUCT
END_TYPE

(* ---- L_MC1P_TRAVERSINGRANGE.dut ---- *)
TYPE L_MC1P_TRAVERSINGRANGE :
(
	MODULO := 0,
	LIMITED := 1
);
END_TYPE

(* ---- L_MC1P_TRCELEMENT.dut ---- *)
TYPE L_MC1P_TRCELEMENT :
STRUCT
	DWCOUNT : DWORD;
	DWTRACEDATA_01 : DWORD;
	DWTRACEDATA_02 : DWORD;
	DWTRACEDATA_03 : DWORD;
	DWTRACEDATA_04 : DWORD;
	DWTRACEDATA_05 : DWORD;
	LRTRACEDATA_06 : LREAL;
	LRTRACEDATA_07 : LREAL;
	LRTRACEDATA_08 : LREAL;
END_STRUCT
END_TYPE

(* ---- L_MC1P_TYPEFUNCTION.dut ---- *)
TYPE L_MC1P_TYPEFUNCTION :
(
	TYPE_ANY := 0,
	TYPE_MC_MOVEABSOLUTE := 10,
	TYPE_MC_MOVEADDITIVE := 20,
	TYPE_MC_MOVECONTINUOUSABSOLUTE := 30,
	TYPE_MC_MOVECONTINUOUSRELATIVE := 40,
	TYPE_MC_MOVERELATIVE := 50,
	TYPE_MC_MOVESUPERIMPOSED := 60,
	TYPE_MC_HALTSUPERIMPOSED := 61,
	TYPE_MC_MOVEVELOCITY := 70,
	TYPE_MC_HALT := 80,
	TYPE_MC_STOP := 90,
	TYPE_MC_CAMIN := 100,
	TYPE_MC_CAMOUT := 110,
	TYPE_MC_GEARIN := 120,
	TYPE_MC_GEARINPOS := 130,
	TYPE_MC_GEAROUT := 140,
	TYPE_MC_COMBINEAXES := 150,
	TYPE_MC_PHASINGRELATIVE := 160,
	TYPE_MC_PHASINGABSOLUTE := 170,
	TYPE_MC_HOME := 180,
	TYPE_MC1P_FOLLOWSETVALUES := 190,
	TYPE_MC1P_TORQUECONTROL := 200,
	TYPE_CT1P_AUTOTUNING := 210
);
END_TYPE

(* ---- L_MC1P_UAXISRETAININFO.dut ---- *)
TYPE L_MC1P_UAXISRETAININFO :
UNION
	INFO : L_MC1P_AxisRetainInfo;
	DWDATA : DWORD;
END_UNION
END_TYPE

(* ---- L_MC1P_UNIVERSALAXISDATATYPES.dut ---- *)
TYPE L_MC1P_UNIVERSALAXISDATATYPES :
UNION
	AXISEXTENSION_I500_CAN : L_MC1P_AxisExtension_i500_CAN;
	AXISEXTENSION_I500_ECAT : L_MC1P_AxisExtension_i500_ECAT;
	AXISEXTENSION_I700 : L_MC1P_AxisExtension_i700;
	AXISEXTENSION_9400HL : L_MC1P_AxisExtension_9400HL;
	AXISEXTENSION_I750 : L_MC1P_AxisExtension_i750;
	AXISEXTENSION_I950 : L_MC1P_AxisExtension_i950;
	AXISEXTENSION_I950_CIAADV : L_MC1P_AxisExtension_i950_CiaAdv;
	AXISEXTENSION_GENERICDRIVE : L_MC1P_AxisExtension_GenericDrive;
END_UNION
END_TYPE

(* ---- L_MC1P_UNIVERSALENCODERDATATYPES.dut ---- *)
TYPE L_MC1P_UNIVERSALENCODERDATATYPES :
UNION
	AXISEXTENSION_ENCFREE : L_MC1P_AxisExtension_EncFree;
	AXISEXTENSION_ENCBPB : L_MC1P_AxisExtension_EncBPB;
	AXISEXTENSION_ENCI500 : L_MC1P_AxisExtension_Enci500;
	AXISEXTENSION_ENCI900_ECAT : L_MC1P_AxisExtension_Enci900_ECAT;
	AXISEXTENSION_ENCIOETC : L_MC1P_AxisExtension_EncIOEtc;
END_UNION
END_TYPE

(* ---- L_MC1P_UNSTEADYREASON.dut ---- *)
TYPE L_MC1P_UNSTEADYREASON :
(
	USRVIRTUAL := 0,
	USRREAL := 1
);
END_TYPE

(* ---- L_MC1P_URETAINDATA.dut ---- *)
TYPE L_MC1P_URETAINDATA :
UNION
	RETAINDATAREALDRIVE : L_MC1P_RetainDataRealDrive_V3;
	RETAINDATAI700 : L_MC1P_RetainDatai700_V3;
END_UNION
END_TYPE

(* ---- L_MC1P_UULINT.dut ---- *)
TYPE L_MC1P_UULINT :
UNION
	ULIDATA : ULINT;
	AUDIDATA : ARRAY [1..2] OF UDINT;
END_UNION
END_TYPE

(* ---- MC_BUFFER_MODE.dut ---- *)
TYPE MC_BUFFER_MODE :
(
	MCABORTING := 0,
	MCBUFFERED := 1,
	MCBLENDINGLOW := 2,
	MCBLENDINGPREVIOUS := 3,
	MCBLENDINGNEXT := 4,
	MCBLENDINGHIGH := 5
);
END_TYPE

(* ---- MC_DIRECTION.dut ---- *)
TYPE MC_DIRECTION :
(
	MCCURRENTDIRECTION := 0,
	MCPOSITIVEDIRECTION := 1,
	MCNEGATIVEDIRECTION := 2,
	MCSHORTESTWAY := 3,
	MCPOSITIVECYCLE := 11,
	MCNEGATIVECYCLE := 12
);
END_TYPE

(* ---- MC_EXECUTION_MODE.dut ---- *)
TYPE MC_EXECUTION_MODE :
(
	MCIMMEDIATELY := 0,
	MCQUEUED := 1
);
END_TYPE

(* ---- MC_SOURCE.dut ---- *)
TYPE MC_SOURCE :
(
	MCSETVALUE := 0,
	MCACTUALVALUE := 1,
	MCCOMMANDEDVALUE := 2
);
END_TYPE

(* ---- MC_TRIGGER_REF.dut ---- *)
TYPE MC_TRIGGER_REF :
STRUCT
	TOUCHPROBESOURCE : BYTE := 1;
	TOUCHPROBECHANNEL : BYTE := 1;
	TOUCHPROBESIGNAL : BYTE := 1;
	TOUCHPROBEEDGE : BYTE := 1;
	TOUCHPROBEMODE : BYTE := 1;
	EXTERNALTPDIGIN : POINTER TO BOOL := 0;
	EXTERNALTPSOURCE : L_IOM_IExternalTPInterface;
	EXTERNALDELAYCOMP : DWORD;
	EXTERNALTPFROMAXIS : L_MC1P_ITPSOURCEAXIS;
	TP_IDENTIFICATION : __XWORD;
END_STRUCT
END_TYPE

(* ---- L_MC1P_CONSTANTS.gvl ---- *)
VAR_GLOBAL
	GC_EPS : LREAL := 1E-10;
	GC_EPS_REAL : LREAL := 1E-06;
	GC_WUPDATEFILTER : WORD := 10;
	GC_WINSTANCENCHAR : WORD := 100;
	GC_WTRACEMAX : WORD := 100;
	GC_IMPLIZITCALLS : INT := 100;
	GC_MAXRETAINAXIS : INT := 256;
	GC_MAXAXISCOUNT : INT := 256;
	GC_ENCFILTERCYCLESMAX : INT := 100;
	GC_DWCHECKIDTAPPETREF : DWORD := 16#DC34;
	GC_SQRT2 : LREAL := 1.4142135623730951;
	GC_PI : LREAL := 3.1415926535897931;
	GC_REC_STATE : LWORD := SHL(1, 0);
	GC_REC_OPMODE : LWORD := SHL(1, 1);
	GC_REC_POS : LWORD := SHL(1, 2);
	GC_REC_VEL : LWORD := SHL(1, 3);
	GC_REC_TORQUE : LWORD := SHL(1, 4);
	GC_REC_ERRORID : LWORD := SHL(1, 5);
	GC_REC_FOLLERROR : LWORD := SHL(1, 6);
	GC_REC_STATELENZE : LWORD := SHL(1, 7);
	GC_REC_STATELENZE2 : LWORD := SHL(1, 8);
	GC_REC_TPSTATE1 : LWORD := SHL(1, 9);
	GC_REC_TP1POS : LWORD := SHL(1, 10);
	GC_REC_TP1NEG : LWORD := SHL(1, 11);
	GC_REC_TP2POS : LWORD := SHL(1, 12);
	GC_REC_TP2NEG : LWORD := SHL(1, 13);
	GC_REC_DIGIN : LWORD := SHL(1, 14);
	GC_REC_STATESM : LWORD := SHL(1, 15);
	GC_REC_VLACTVELOCITY : LWORD := SHL(1, 16);
	GC_REC_ENCPOS : LWORD := SHL(1, 17);
	GC_REC_ENCVEL : LWORD := SHL(1, 18);
	GC_REC_TP1POSTIME : LWORD := SHL(1, 19);
	GC_REC_TP1NEGTIME : LWORD := SHL(1, 20);
	GC_REC_TP2POSTIME : LWORD := SHL(1, 21);
	GC_REC_TP2NEGTIME : LWORD := SHL(1, 22);
	GC_REC_TPSTATE2 : LWORD := SHL(1, 23);
	GC_REC_TP3POS : LWORD := SHL(1, 24);
	GC_REC_TP3NEG : LWORD := SHL(1, 25);
	GC_REC_TP4POS : LWORD := SHL(1, 26);
	GC_REC_TP4NEG : LWORD := SHL(1, 27);
	GC_REC_TP3POSTIME : LWORD := SHL(1, 28);
	GC_REC_TP3NEGTIME : LWORD := SHL(1, 29);
	GC_REC_TP4POSTIME : LWORD := SHL(1, 30);
	GC_REC_TP4NEGTIME : LWORD := SHL(1, 31);
	GC_REC_SAFETYCTRL : LWORD := SHL(1, 32);
	GC_REC_SAFETYSTATE : LWORD := SHL(1, 33);
	GC_REC_SAFETYIOSTATE : LWORD := SHL(1, 34);
	GC_REC_ENCPOSTIMESTAMP : LWORD := SHL(1, 35);
	GC_REC_STATELENZEEXT : LWORD := SHL(1, 36);
	GC_REC_SPEEDERROR : LWORD := SHL(1, 37);
	GC_REC_POSVALUE1616 : LWORD := SHL(1, 38);
	GC_REC_CONTROLEFFORT : LWORD := SHL(1, 39);
	GC_REC_ACTPOSMOTORCIA402ADV : LWORD := SHL(1, 40);
	GC_REC_TEXTREFID : LWORD := SHL(1, 41);
	GC_REC_POSTIMESTAMP : LWORD := SHL(1, 42);
	GC_REC_MAXDATAINDEX : WORD := 43;
	GC_TRANS_CTRL : LWORD := SHL(1, 0);
	GC_TRANS_OPMODE : LWORD := SHL(1, 1);
	GC_TRANS_POS : LWORD := SHL(1, 2);
	GC_TRANS_VEL : LWORD := SHL(1, 3);
	GC_TRANS_TORQUE : LWORD := SHL(1, 4);
	GC_TRANS_TORQUELIMPOS : LWORD := SHL(1, 5);
	GC_TRANS_TORQUELIMNEG : LWORD := SHL(1, 6);
	GC_TRANS_SPEEDLIMUP : LWORD := SHL(1, 7);
	GC_TRANS_SPEEDLIMLOW : LWORD := SHL(1, 8);
	GC_TRANS_TPCTRL1 : LWORD := SHL(1, 9);
	GC_TRANS_POSOFFSET : LWORD := SHL(1, 10);
	GC_TRANS_VELOFFSET : LWORD := SHL(1, 11);
	GC_TRANS_TORQUEOFFSET : LWORD := SHL(1, 12);
	GC_TRANS_SPEEDCTRLINT : LWORD := SHL(1, 13);
	GC_TRANS_CTRLLENZE : LWORD := SHL(1, 14);
	GC_TRANS_VLTARGETVELOCITY : LWORD := SHL(1, 16);
	GC_TRANS_BRKOVRD : LWORD := SHL(1, 17);
	GC_TRANS_CTRLLENZE2 : LWORD := SHL(1, 18);
	GC_TRANS_CTRLLENZE3 : LWORD := SHL(1, 19);
	GC_TRANS_CTRLLENZE4 : LWORD := SHL(1, 20);
	GC_TRANS_TPCTRL2 : LWORD := SHL(1, 21);
	GC_TRANS_SAFEPOS : LWORD := SHL(1, 22);
	GC_TRANS_SAFEPOSSTATUS : LWORD := SHL(1, 23);
	GC_TRANS_SPEEDLIMITSLS : LWORD := SHL(1, 24);
	GC_TRANS_MAXDATAINDEX : WORD := 25;
	NODATAMEMORYAVAILABLE : WORD := WORD#16#1;
	MEMORYINVALID : WORD := WORD#16#2;
	MEMORYNOTINITIALIZED : WORD := WORD#16#4;
	NODATAAVAILABLE : WORD := WORD#16#8;
	NOMEMORYAVAILABLEFORAXIS : WORD := WORD#16#10;
	NOMEMORYINAXISARRAY : WORD := WORD#16#20;
	AXISGUIDCHANGED : WORD := WORD#16#40;
	C_SERIALNUMBER : UINT := 3;
	C_MANUFACTURER : UINT := 5;
	C_SOFTWAREREVISION : UINT := 9;
	C_HARDWAREREVISION : UINT := 10;
	C_DEVICECLASS : UINT := 11;
	C_PRODUCTCODE : UINT := 13;
	C_UPDATE : UINT := 99;
	C_CONNECTORTYPEMOTIONAXISOLD : UINT := 1279;
	C_CONNECTORTYPEMOTIONAXIS : UINT := 34279;
	C_CONNECTORTYPEENCODERIOSLICE : UINT := 33024;
END_VAR

(* ---- L_MC1P_INTERNAL.gvl ---- *)
VAR_GLOBAL
	DWDUMMY : DWORD;
	XAPPFIRSTRUN : BOOL := FALSE;
	PANYCONNECTOR : POINTER TO IoConfigConnector;
	LMAXISRETAINHANDLING : L_MC1P_AxisRetainMangaement;
	DWTIMESTAMPSIMU : DWORD;
	XTIMESTAMPUPDATED : BOOL;
	LMAXISMGMT : L_MC1P_AxisManagementFunction;
	CDIENUMSTARTVALUE : DINT := 50000;
END_VAR

(* ---- L_MC1P_IAXIS_REF_BRAKE.itf ---- *)
INTERFACE L_MC1P_IAXIS_REF_BRAKE
END_INTERFACE

METHOD GETACTVALUESBRAKE
END_METHOD

METHOD SWITCHONCONTROL
VAR_INPUT
	XSWITCHONREQUEST : BOOL;
END_VAR
VAR_OUTPUT
	XSWITCHON : BOOL;
END_VAR
VAR_IN_OUT
	AXIS : AXIS_REF;
END_VAR
END_METHOD

METHOD SWITCHEDONSTATUS
VAR_INPUT
	XSWITCHEDONREQUEST : BOOL;
END_VAR
VAR_OUTPUT
	XSWITCHEDON : BOOL;
END_VAR
VAR_IN_OUT
	AXIS : AXIS_REF;
END_VAR
END_METHOD

(* ---- L_MC1P_IAXIS_REF_MASTERVALUES.itf ---- *)
INTERFACE L_MC1P_IAXIS_REF_MASTERVALUES
END_INTERFACE

METHOD GETDIRECTION : WORD
VAR_INPUT
	VALUESOURCE : MC_SOURCE;
END_VAR
END_METHOD

METHOD GETMASTERERROR : BOOL
VAR_OUTPUT
	EERRORID : L_IE1P_Error;
END_VAR
END_METHOD

METHOD GETSTEADYSTATE : POINTER TO L_MC1P_SteadyState
END_METHOD

(* ---- L_MC1P_IAXIS_REF_POOL.itf ---- *)
INTERFACE L_MC1P_IAXIS_REF_POOL
END_INTERFACE

METHOD GETAXISFROMPOOL : POINTER TO AXIS_REF
VAR_INPUT
	WINDEX : WORD;
END_VAR
END_METHOD

(* ---- L_MC1P_IAXISCOMMMAND.itf ---- *)
INTERFACE L_MC1P_IAXISCOMMMAND
END_INTERFACE

METHOD ABORTING
END_METHOD

METHOD CALCSTATUS
VAR_IN_OUT
	AXIS : _AXIS_REF_REAL;
END_VAR
END_METHOD

METHOD EXECUTE
END_METHOD

METHOD MAIN
END_METHOD

METHOD RESETCOMMANDERRORSTATE : BOOL
VAR_IN_OUT
	AXIS : _AXIS_REF_REAL;
END_VAR
END_METHOD

METHOD RESETSTATUSPARAMETER
END_METHOD

METHOD SETINCTANCEINFO
VAR_INPUT
	PSINSTANCENAME : POINTER TO STRING;
	ERRORITFID : DWORD;
END_VAR
END_METHOD

METHOD UPDATEAXISPOINTER
VAR_INPUT
	PAXIS : POINTER TO AXIS_REF;
END_VAR
END_METHOD

METHOD UPDATECOMMANDINTERFACE
VAR_IN_OUT
	CMD : USINT;
END_VAR
END_METHOD

(* ---- L_MC1P_IAXISCOMMMAND_AUTOTUNING.itf ---- *)
INTERFACE L_MC1P_IAXISCOMMMAND_AUTOTUNING
END_INTERFACE

METHOD CALCPROFILEPARAMS
VAR_IN_OUT
	AXIS : AXIS_REF;
END_VAR
END_METHOD

METHOD UPDATEPARAINTERFACE
VAR_IN_OUT
	SCPAR : L_MC1P_AutotuningPara;
END_VAR
END_METHOD

(* ---- L_MC1P_IAXISEXTENSION.itf ---- *)
INTERFACE L_MC1P_IAXISEXTENSION
END_INTERFACE

METHOD SETBASICINITIALISATION
VAR_INPUT
	ITFGENERICCONFIG : L_MC1P_IGenericAxisConfiguration;
END_VAR
VAR_IN_OUT
	AXIS : _AXIS_REF_REAL;
END_VAR
END_METHOD

(* ---- L_MC1P_IAXISSIMULATIONINTERFACE.itf ---- *)
INTERFACE L_MC1P_IAXISSIMULATIONINTERFACE
END_INTERFACE

METHOD ACTIVATESIMULATION
VAR_IN_OUT
	AXIS : _AXIS_REF_REAL;
END_VAR
END_METHOD

METHOD CALCULATEINPUTDATA
VAR_IN_OUT
	AXIS : _AXIS_REF_REAL;
END_VAR
END_METHOD

METHOD CALCULATEOUTPUTDATA
VAR_IN_OUT
	AXIS : _AXIS_REF_REAL;
END_VAR
END_METHOD

METHOD DISABLESIMULATION
VAR_IN_OUT
	AXIS : _AXIS_REF_REAL;
END_VAR
END_METHOD

(* ---- L_MC1P_ICOMMMUNICATIONSIMULATION.itf ---- *)
INTERFACE L_MC1P_ICOMMMUNICATIONSIMULATION
END_INTERFACE

METHOD GETCOMMSTATE : L_DCO_CommState
VAR_INPUT
	PAXISCOMM : POINTER TO _AXIS_REF_COM;
END_VAR
END_METHOD

METHOD PARREAD
VAR_INPUT
	WIDX : DWORD;
END_VAR
END_METHOD

METHOD PARREAD_GETOUTPUT
VAR_INPUT
	WIDX : DWORD;
END_VAR
VAR_OUTPUT
	SZDATAREAD : CAA_SIZE;
	XDONE : BOOL;
	XERROR : BOOL;
	WERROR : WORD;
END_VAR
END_METHOD

METHOD PARREAD_SETINPUT
VAR_INPUT
	WIDX : DWORD;
	XEXECUTE : BOOL;
	WINDEX : WORD;
	BYSUBINDEX : BYTE;
	PBUFFER : POINTER TO BYTE;
	SZSIZE : UDINT;
	UDITIMEOUT : UDINT;
	XSLOTB : BOOL;
END_VAR
END_METHOD

METHOD PARWRITE
VAR_INPUT
	WIDX : DWORD;
END_VAR
END_METHOD

METHOD PARWRITE_GETOUTPUT
VAR_INPUT
	WIDX : DWORD;
END_VAR
VAR_OUTPUT
	XDONE : BOOL;
	XERROR : BOOL;
	WERROR : WORD;
END_VAR
END_METHOD

METHOD PARWRITE_SETINPUT
VAR_INPUT
	WIDX : DWORD;
	XEXECUTE : BOOL;
	WINDEX : WORD;
	BYSUBINDEX : BYTE;
	PBUFFER : POINTER TO BYTE;
	SZSIZE : UDINT;
	UDITIMEOUT : UDINT;
	XSLOTB : BOOL;
END_VAR
END_METHOD

METHOD RESTARTMASTER
VAR_INPUT
	XEXECUTE : BOOL;
	PAXIS : POINTER TO _AXIS_REF_COM;
END_VAR
VAR_OUTPUT
	XDONE : BOOL;
	XERROR : BOOL;
	XBUSY : BOOL;
	DWERROR : DWORD;
END_VAR
END_METHOD

(* ---- L_MC1P_ICOMMUNICATION.itf ---- *)
INTERFACE L_MC1P_ICOMMUNICATION
END_INTERFACE

METHOD FORWARDERROR
VAR_INPUT
	XENABLE : BOOL;
	XWARNING : BOOL;
	XERROR : BOOL;
	WERRORID : WORD;
	WTEXTREFID : WORD;
	XRESETERROR : BOOL := FALSE;
	AXISMODULEHANDLER : L_IMHP_IModuleHandler;
END_VAR
END_METHOD

METHOD GETCOMMPARAMETER
VAR_INPUT
	PCONNECTOR : POINTER TO IoConfigConnector;
END_VAR
VAR_OUTPUT
	PSLAVECONNECTOR : POINTER TO IoStandard.IoConfigConnector;
	UINETID : UINT;
	UIDEVICEID : UINT;
	XSENDFRAMEATTASKSTART : BOOL;
	UDIPRODUCTCODE : DWORD;
	PMASTERCONNECTOR : POINTER TO IoStandard.IoConfigConnector;
END_VAR
END_METHOD

METHOD GETCOMMSTATE : L_DCO_CommState
VAR_INPUT
	PAXISCOMM : POINTER TO _AXIS_REF_COM;
END_VAR
END_METHOD

METHOD GETPDINEQPDOUT : BOOL
END_METHOD

METHOD PARREAD
VAR_INPUT
	WIDX : DWORD;
END_VAR
END_METHOD

METHOD PARREAD_GETOUTPUT
VAR_INPUT
	WIDX : DWORD;
END_VAR
VAR_OUTPUT
	SZDATAREAD : CAA_SIZE;
	XDONE : BOOL;
	XERROR : BOOL;
	WERROR : WORD;
END_VAR
END_METHOD

METHOD PARREAD_SETINPUT
VAR_INPUT
	WIDX : DWORD;
	XEXECUTE : BOOL;
	WINDEX : WORD;
	BYSUBINDEX : BYTE;
	PBUFFER : POINTER TO BYTE;
	SZSIZE : UDINT;
	UDITIMEOUT : UDINT;
END_VAR
END_METHOD

METHOD PARWRITE
VAR_INPUT
	WIDX : DWORD;
END_VAR
END_METHOD

METHOD PARWRITE_GETOUTPUT
VAR_INPUT
	WIDX : DWORD;
END_VAR
VAR_OUTPUT
	XDONE : BOOL;
	XERROR : BOOL;
	WERROR : WORD;
END_VAR
END_METHOD

METHOD PARWRITE_SETINPUT
VAR_INPUT
	WIDX : DWORD;
	XEXECUTE : BOOL;
	WINDEX : WORD;
	BYSUBINDEX : BYTE;
	PBUFFER : POINTER TO BYTE;
	SZSIZE : UDINT;
	UDITIMEOUT : UDINT;
END_VAR
END_METHOD

METHOD RESET
END_METHOD

METHOD RESTARTMASTER
VAR_INPUT
	XEXECUTE : BOOL;
	PAXIS : POINTER TO _AXIS_REF_COM;
END_VAR
VAR_OUTPUT
	XDONE : BOOL;
	XERROR : BOOL;
	XBUSY : BOOL;
	DWERROR : DWORD;
END_VAR
END_METHOD

METHOD SETBASICINITIALISATION
VAR_IN_OUT
	AXIS : _AXIS_REF_REAL;
END_VAR
END_METHOD

METHOD SETCOMPONENTINFO
VAR_INPUT
	DATASELECTION : WORD;
	SDATA : STRING;
END_VAR
END_METHOD

(* ---- L_MC1P_ICOMPENSATIONINTERFACE.itf ---- *)
INTERFACE L_MC1P_ICOMPENSATIONINTERFACE
END_INTERFACE

METHOD GETOFFSETVALUES
VAR_OUTPUT
	LROFFSETPOS : LREAL;
	LROFFSETVEL : LREAL;
	LROFFSETACC : LREAL;
END_VAR
END_METHOD

(* ---- L_MC1P_ICONFIGUREDRIVE.itf ---- *)
INTERFACE L_MC1P_ICONFIGUREDRIVE
END_INTERFACE

METHOD DOFUNCTION : BOOL
VAR_INPUT
	XEXECUTE : BOOL;
	WOFFSET : WORD;
END_VAR
VAR_OUTPUT
	XDONE : BOOL;
	XERROR : BOOL;
	XBUSY : BOOL;
	EERRORID : WORD;
END_VAR
VAR_IN_OUT
	AXIS : _AXIS_REF_REAL;
END_VAR
END_METHOD

METHOD GETADDITIONALCONFIGINFO : POINTER TO L_MC1P_AdditionalConfigInfo
END_METHOD

METHOD GETINSTANCE : POINTER TO BYTE
END_METHOD

METHOD RESET : BOOL
END_METHOD

(* ---- L_MC1P_ICONTROLLERADAPTION.itf ---- *)
INTERFACE L_MC1P_ICONTROLLERADAPTION
END_INTERFACE

METHOD CALCADAPTIONCURVE : LREAL
VAR_INPUT
	LRSETVEL : LREAL;
END_VAR
VAR_IN_OUT
	AXIS : _AXIS_REF_REAL;
END_VAR
END_METHOD

(* ---- L_MC1P_ICONTROLLERINTERFACE.itf ---- *)
INTERFACE L_MC1P_ICONTROLLERINTERFACE
END_INTERFACE

METHOD CALCCONTROLLER
VAR_INPUT
	LRSETPOSITION : LREAL;
	LRSETVELOCITY : LREAL;
	LRSETACCELERATION : LREAL;
	LRSETTORQUE : LREAL;
	LRSETJERK : LREAL;
	LRACTPOSITIONIN : LREAL;
	LRACTVELOCITYIN : LREAL;
	LRACTACCELERATIONIN : LREAL;
	LRACTTORQUEIN : LREAL;
END_VAR
VAR_OUTPUT
	LRSETPOSITIONOUT : LREAL;
	LRSETVELOCITYOUT : LREAL;
	LRSETACCELERATIONOUT : LREAL;
	LRSETTORQUEOUT : LREAL;
END_VAR
VAR_IN_OUT
	AXIS : _AXIS_REF_REAL;
END_VAR
END_METHOD

(* ---- L_MC1P_IDRIVESCALING.itf ---- *)
INTERFACE L_MC1P_IDRIVESCALING
END_INTERFACE

METHOD CALCACCFACTOR : BOOL
VAR_OUTPUT
	LRSCALEUNITTOACC : LREAL;
	LRSCALEACCTOUNIT : LREAL;
END_VAR
VAR_IN_OUT
	AXIS : _AXIS_REF_REAL;
END_VAR
END_METHOD

METHOD CALCSPEEDFACTOR : BOOL
VAR_OUTPUT
	LRSCALEUNITTOSPEED : LREAL;
	LRSCALESPEEDTOUNIT : LREAL;
END_VAR
VAR_IN_OUT
	AXIS : _AXIS_REF_REAL;
END_VAR
END_METHOD

METHOD CALCTORQUEFACTOR : BOOL
VAR_OUTPUT
	LRSCALETORQUETONORM : LREAL;
	LRSCALETORQUETONORM2 : LREAL;
	LRSCALENORMTOTORQUE : LREAL;
END_VAR
VAR_IN_OUT
	AXIS : _AXIS_REF_REAL;
END_VAR
END_METHOD

METHOD CHECKVALIDPOSRESOLUTION : BOOL
VAR_INPUT
	DWPOSRESOLUTION : DWORD;
END_VAR
END_METHOD

METHOD GETDEFAULTTORQUE : LREAL
VAR_INPUT
	LRREFTORQUE : LREAL;
END_VAR
END_METHOD

METHOD POSDIFFTOSPEEDINC : DINT
VAR_INPUT
	DIPOSDIFF : DINT := 0;
	DWFACTOR : DWORD := 1000;
END_VAR
VAR_IN_OUT
	AXIS : _AXIS_REF_REAL;
END_VAR
END_METHOD

METHOD SPEEDTOPOSDIFFINC : DINT
VAR_INPUT
	DISPEED : DINT := 0;
	DWFACTOR : DWORD := 1000;
END_VAR
VAR_IN_OUT
	AXIS : _AXIS_REF_REAL;
	DIRES : DINT;
END_VAR
END_METHOD

(* ---- L_MC1P_IDRIVESPECIFICIMPLBASE.itf ---- *)
INTERFACE L_MC1P_IDRIVESPECIFICIMPLBASE
END_INTERFACE

METHOD CALCAFTERREADINPUTS
VAR_IN_OUT
	AXIS : _AXIS_REF_REAL;
END_VAR
END_METHOD

METHOD CALCBEFOREREADINPUTS
VAR_IN_OUT
	AXIS : _AXIS_REF_REAL;
END_VAR
END_METHOD

METHOD CALCBEFOREWRITEOUTPUTS
VAR_IN_OUT
	AXIS : _AXIS_REF_REAL;
END_VAR
END_METHOD

METHOD CHECKAVAILABLECONTROLMODE : BOOL
VAR_IN_OUT
	AXIS : _AXIS_REF_REAL;
	POSCTRLDRIVEAVAILABLE : L_IE1P_Error;
	POSCTRLPLCAVAILABLE : L_IE1P_Error;
	SPEEDCTRLDRIVEAVAILABLE : L_IE1P_Error;
	TORQUECTRLDRIVE : L_IE1P_Error;
END_VAR
END_METHOD

METHOD CHECKRESETHOMEPOS
VAR_INPUT
	WFDBSTATUSWORD : WORD;
END_VAR
VAR_IN_OUT
	AXIS : _AXIS_REF_REAL;
END_VAR
END_METHOD

METHOD CHECKSAFETYOPTIONAVAILABLE : BOOL
VAR_INPUT
	DWPRODUCTCODE : DWORD;
END_VAR
END_METHOD

METHOD COLLECTDRIVESTATE : BOOL
VAR_IN_OUT
	AXIS : _AXIS_REF_REAL;
	SCSTATEINFO : L_MC1P_DriveStateCollection;
END_VAR
END_METHOD

METHOD CONTROLDRIVE : BOOL
VAR_INPUT
	XENABLE : BOOL;
END_VAR
VAR_IN_OUT
	AXIS : _AXIS_REF_REAL;
END_VAR
END_METHOD

METHOD DRIVECONFIGDATA
VAR_INPUT
	PCONFIGINFO : POINTER TO L_MC1P_AdditionalConfigInfo;
END_VAR
VAR_IN_OUT
	AXIS : _AXIS_REF_REAL;
END_VAR
END_METHOD

METHOD DRIVEFAULTSTATUS : BOOL
VAR_IN_OUT
	AXIS : _AXIS_REF_REAL;
	SCSTATEINFO : L_MC1P_DriveStateCollection;
END_VAR
END_METHOD

METHOD GETBRAKE : POINTER TO L_MC1P_BrakeControlBase
VAR_IN_OUT
	AXIS : _AXIS_REF_REAL;
END_VAR
END_METHOD

METHOD GETBRAKESERVICE : POINTER TO L_MC1P_BrakeService
VAR_IN_OUT
	AXIS : _AXIS_REF_REAL;
END_VAR
END_METHOD

METHOD GETCAUSEOFCINH : WORD
VAR_IN_OUT
	AXIS : _AXIS_REF_REAL;
END_VAR
END_METHOD

METHOD GETFDBSTATUSWORD : WORD
VAR_IN_OUT
	AXIS : _AXIS_REF_REAL;
END_VAR
END_METHOD

METHOD GETIECADRESS : BOOL
VAR_IN_OUT
	AXIS : _AXIS_REF_REAL;
	M_PPDOINFOCONNECTOR : POINTER TO IoConfigConnector;
	ATRANSELEMENT : ARRAY [1.._AXIS_REF_REAL.c_wMaxTransElem] OF L_MC1P_MappedElement;
	WTRANSELEMENTS : WORD;
	LWTRANSDATA : LWORD;
	LWRECDATA : LWORD;
	WRECEIVEELEMENTS : WORD;
	ARECEIVEELEMENT : ARRAY [1.._AXIS_REF_REAL.c_wMaxRecElem] OF L_MC1P_MappedElement;
END_VAR
END_METHOD

METHOD GETOPTIONALACTVEL : BOOL
VAR_IN_OUT
	LRVEL : LREAL;
END_VAR
END_METHOD

METHOD GETRECEIVEDATAIMPL : DWORD
VAR_INPUT
	LWMASK : LWORD;
END_VAR
VAR_IN_OUT
	AXIS : _AXIS_REF_REAL;
END_VAR
END_METHOD

METHOD GETSTATUSWORDS
VAR_OUTPUT
	STATUSWORD1 : WORD;
	STATUSWORD2 : WORD;
	STATUSWORD3 : WORD;
	STATUSWORD4 : WORD;
END_VAR
VAR_IN_OUT
	AXIS : _AXIS_REF_REAL;
END_VAR
END_METHOD

METHOD GETTRANSMITDATAIMPL : DWORD
VAR_INPUT
	LWMASK : LWORD;
END_VAR
VAR_IN_OUT
	AXIS : _AXIS_REF_REAL;
END_VAR
END_METHOD

METHOD GETTRANSMITDATALREALIMPL : LREAL
VAR_INPUT
	LWMASK : LWORD;
END_VAR
VAR_IN_OUT
	AXIS : _AXIS_REF_REAL;
END_VAR
END_METHOD

METHOD HOMECONFIG : BOOL
VAR_INPUT
	LRPOSITION : LREAL;
END_VAR
VAR_OUTPUT
	WINDEX : WORD;
	BYSUBINDEX : BYTE;
	BYNROFBYTE : BYTE;
	DWDATA : DWORD;
	XWRITEPARAM : BOOL;
	XDONE : BOOL;
	XERROR : BOOL;
END_VAR
VAR_IN_OUT
	AXIS : _AXIS_REF_REAL;
	SCHOMEDATA : L_MC1P_HomeParameter;
	WSTEP : WORD;
END_VAR
END_METHOD

METHOD HOMEPOSPERMANENTSETACTIVE : BOOL
VAR_IN_OUT
	AXIS : _AXIS_REF_REAL;
END_VAR
END_METHOD

METHOD RECEIVEPARAMETER
VAR_INPUT
	WPARAMETER : WORD;
	PADRESS : POINTER TO BYTE;
	WSIZE : WORD;
END_VAR
VAR_IN_OUT
	AXIS : _AXIS_REF_REAL;
END_VAR
END_METHOD

METHOD RECEIVEPARAMETERCALC
VAR_IN_OUT
	AXIS : _AXIS_REF_REAL;
	DATA : ARRAY [1..L_MC1P_Constants.gc_Rec_MaxDataIndex] OF POINTER TO L_MC1P_MappedElement;
END_VAR
END_METHOD

METHOD RESETDRIVECONTROL
VAR_INPUT
	XRESETDRIVEERROR : BOOL;
END_VAR
END_METHOD

METHOD RESTOREADDITIONALRETAINDATA
VAR_INPUT
	PDATA : POINTER TO L_MC1P_uRetainData;
END_VAR
END_METHOD

METHOD SETAXISPROPERTIES
VAR_IN_OUT
	AXIS : _AXIS_REF_REAL;
	AXISPROPERTIES : L_MC1P_AxisProperties;
END_VAR
END_METHOD

METHOD SETAXISSTATUSWORD
VAR_IN_OUT
	AXIS : _AXIS_REF_REAL;
	DWAXISSTATUS : DWORD;
END_VAR
END_METHOD

METHOD SETBASICINITIALISATION
VAR_IN_OUT
	AXIS : _AXIS_REF_REAL;
END_VAR
END_METHOD

METHOD SETCONTROLWORDS
VAR_INPUT
	CONTROLWORD1 : WORD;
	CONTROLWORD2 : WORD;
	CONTROLWORD3 : WORD;
	CONTROLWORD4 : WORD;
END_VAR
VAR_IN_OUT
	AXIS : _AXIS_REF_REAL;
END_VAR
END_METHOD

METHOD SETDCBRAKE
VAR_INPUT
	XSETDCBRAKE : BOOL;
END_VAR
VAR_OUTPUT
	XDCBRAKEACTIVE : BOOL;
END_VAR
VAR_IN_OUT
	AXIS : _AXIS_REF_REAL;
END_VAR
END_METHOD

METHOD SETDRIVECONFIGINIT
VAR_IN_OUT
	AXIS : _AXIS_REF_REAL;
END_VAR
END_METHOD

METHOD SETSPEEDCTRLLIMITATION : BOOL
VAR_INPUT
	XLIMIT : BOOL;
END_VAR
VAR_IN_OUT
	AXIS : _AXIS_REF_REAL;
END_VAR
END_METHOD

METHOD SETSPEEDCTRLLOADVALUE
VAR_INPUT
	XLOAD : BOOL;
	LRVALUE : LREAL;
END_VAR
VAR_IN_OUT
	AXIS : _AXIS_REF_REAL;
END_VAR
END_METHOD

METHOD STOREADDITIONALRETAINDATA
VAR_INPUT
	PDATA : POINTER TO L_MC1P_uRetainData;
END_VAR
END_METHOD

METHOD TRANSMITPARAMETER
VAR_INPUT
	WPARAMETER : WORD;
	PADRESS : POINTER TO BYTE;
	WSIZE : WORD;
END_VAR
VAR_IN_OUT
	AXIS : _AXIS_REF_REAL;
END_VAR
END_METHOD

METHOD TRANSMITPARAMETERCALC
VAR_IN_OUT
	AXIS : _AXIS_REF_REAL;
	DATA : ARRAY [1..L_MC1P_Constants.gc_Trans_MaxDataIndex] OF POINTER TO L_MC1P_MappedElement;
END_VAR
END_METHOD

METHOD UPDATEMAPPING
VAR_INPUT
	PTASKMAPLIST : POINTER TO IoStandard.IoConfigTaskMap;
	NCOUNT : DINT;
	PPDOINFOCONNECTOR : POINTER TO IoConfigConnector;
END_VAR
VAR_IN_OUT
	AXIS : _AXIS_REF_REAL;
END_VAR
END_METHOD

(* ---- L_MC1P_IDRIVEUTILS.itf ---- *)
INTERFACE L_MC1P_IDRIVEUTILS
END_INTERFACE

METHOD ACTIVATEAPPCREDITS
VAR_INPUT
	XACTIVATE : BOOL;
END_VAR
END_METHOD

METHOD GETMULTIAXISINFO
VAR_IN_OUT
	MULTIAXISINFO : L_MC1P_MultiAxisInfo;
END_VAR
END_METHOD

METHOD GETRETAINMEMINFO : L_MC1P_RetainDataType
VAR_OUTPUT
	MEMINFO : L_MC1P_uAxisRetainInfo;
END_VAR
END_METHOD

METHOD RESETCONNECTION : L_IE1P_Error
VAR_INPUT
	ITFCALLEDFUNCITON : L_IF1P_IFunctionConnection;
	EDISCONNECTMODE : L_IF1P_DisconnectMode;
	XDISCONNECTEXISTINGCONNECTION : BOOL;
END_VAR
END_METHOD

METHOD SETCONNECTION
VAR_INPUT
	AXISCONNECTION : L_IF1P_IFunctionConnection;
END_VAR
END_METHOD

(* ---- L_MC1P_IENCODERINTERFACE.itf ---- *)
INTERFACE L_MC1P_IENCODERINTERFACE
END_INTERFACE

METHOD ENCNEWHOMEPOSLOADED : BOOL
VAR_INPUT
	DWCALLYCLE : DWORD;
	DWDELAY : DWORD;
END_VAR
END_METHOD

METHOD ENCRESETACTPOS
END_METHOD

METHOD ENCRESETHOMEPOS
VAR_INPUT
	ERESETINFO : L_IE1P_Error;
END_VAR
END_METHOD

METHOD ENCSETHOMEPOSITION
VAR_INPUT
	POSITION : LREAL;
	RELATIVE : BOOL;
	POSDIFF : LREAL;
	EHOMEPOSINFO : L_IE1P_Error;
END_VAR
END_METHOD

METHOD ENCSIGNALVALID : BOOL
VAR_OUTPUT
	XSIGNALVALIDOLD : BOOL;
	EENCERRORID : L_IE1P_Error;
END_VAR
END_METHOD

METHOD GETACTPOSINCR : DINT
END_METHOD

METHOD GETACTPOSINCR1616 : DINT
END_METHOD

METHOD GETACTVALUES
VAR_OUTPUT
	LRACTPOS : LREAL;
	LRACTVEL : LREAL;
	LRACTACC : LREAL;
	LRACTPOSUNFILTERED : LREAL;
	LRACTPOSROUNDS : LREAL;
END_VAR
END_METHOD

METHOD GETAXISINSTANCE : POINTER TO _AXIS_REF_REAL
END_METHOD

METHOD GETCONFIGCHANGED : BOOL
END_METHOD

METHOD GETHOMEPOSAVAILABLE : BOOL
END_METHOD

METHOD SETHOMEPOSAVAILABLE
VAR_INPUT
	XHOMEPOSAVAILABLE : BOOL;
END_VAR
END_METHOD

(* ---- L_MC1P_IENCODERPOSFILTER.itf ---- *)
INTERFACE L_MC1P_IENCODERPOSFILTER
END_INTERFACE

METHOD CALCULATE
VAR_INPUT
	LRCYCPOSIN : LREAL;
	LRCYCVELIN : LREAL;
END_VAR
VAR_OUTPUT
	LRCYCPOSOUT : LREAL;
	LRCYCVELOUT : LREAL;
	WFILTERSTATE : WORD;
END_VAR
END_METHOD

METHOD INIT
END_METHOD

METHOD RESET
END_METHOD

(* ---- L_MC1P_IEXTENDEDMAPPINGACCESS.itf ---- *)
INTERFACE L_MC1P_IEXTENDEDMAPPINGACCESS
END_INTERFACE

METHOD GETIECADRESS
VAR_INPUT
	AXISCONNECTOR : POINTER TO IoConfigConnector;
END_VAR
END_METHOD

METHOD GETMAPPEDDATA : POINTER TO BYTE
VAR_INPUT
	UIINDEX : WORD;
	USISUBINDEX : USINT;
	USISIZE : USINT;
	XWRITEACCESS : BOOL;
	PADDDATA : POINTER TO BYTE;
	PXWAITFORINITACCESS : POINTER TO BOOL;
END_VAR
VAR_OUTPUT
	EERRORID : L_IE1P_Error;
	XERROR : BOOL;
	USISIZEACT : USINT;
END_VAR
END_METHOD

METHOD GETMAPPEDDATASUPPORT : BOOL
END_METHOD

METHOD RESETOUTPUTMAPPINGOBJECTS : BOOL
END_METHOD

(* ---- L_MC1P_IGENERICAXISCONFIGURATION.itf ---- *)
INTERFACE L_MC1P_IGENERICAXISCONFIGURATION
END_INTERFACE

METHOD CALCAFTERREADINPUTS
VAR_IN_OUT
	AXIS : _AXIS_REF_REAL;
	DRIVESPECIFIC : L_MC1P_DriveSpecific_Generic;
END_VAR
END_METHOD

METHOD CALCBEFOREREADINPUTS
VAR_IN_OUT
	AXIS : _AXIS_REF_REAL;
	DRIVESPECIFIC : L_MC1P_DriveSpecific_Generic;
END_VAR
END_METHOD

METHOD CALCBEFOREWRITEOUTPUTS
VAR_IN_OUT
	AXIS : _AXIS_REF_REAL;
	DRIVESPECIFIC : L_MC1P_DriveSpecific_Generic;
END_VAR
END_METHOD

METHOD DRIVECONFIG
VAR_INPUT
	WOFFSET : WORD;
END_VAR
VAR_OUTPUT
	XCONFIGBUSY : BOOL;
	XWAITFORPARAMETERWRITEDONE : BOOL;
	XWAITFORPARAMETERREADDONE : BOOL;
	XREADSTRING : BOOL;
	DWWRITEDATA : DWORD;
	WINDEX : WORD;
	BYSUBINDEX : BYTE;
	BYNROFBYTE : BYTE;
END_VAR
VAR_IN_OUT
	AXIS : _AXIS_REF_REAL;
	CONFIGINFO : L_MC1P_AdditionalConfigInfo;
	WSTEP : WORD;
	EERRORID : WORD;
	DWREADDATA : DWORD;
	SREADDATA : STRING(255);
END_VAR
END_METHOD

METHOD GETADDITIONALSTATEINFOS : BOOL
VAR_IN_OUT
	AXIS : _AXIS_REF_REAL;
	DRIVESPECIFIC : L_MC1P_DriveSpecific_Generic;
	SCSTATEINFO : L_MC1P_DriveStateCollection;
END_VAR
END_METHOD

METHOD GETHOMINGSTATE
VAR_INPUT
	WHOMESTATE : WORD;
END_VAR
VAR_IN_OUT
	AXIS : _AXIS_REF_REAL;
	XHOMEPOSAVAILABLEDRIVE : BOOL;
END_VAR
END_METHOD

METHOD HOMECONFIG
VAR_INPUT
	LRPOSITION : LREAL;
END_VAR
VAR_OUTPUT
	XCONFIGBUSY : BOOL;
	XERROR : BOOL;
	WINDEX : WORD;
	BYSUBINDEX : BYTE;
	BYNROFBYTE : BYTE;
	DWDATA : DWORD;
	XWRITEPARAM : BOOL;
END_VAR
VAR_IN_OUT
	AXIS : _AXIS_REF_REAL;
	SCHOMEDATA : L_MC1P_HomeParameter;
	WSTEP : WORD;
END_VAR
END_METHOD

METHOD RECEIVEPARAMETERCALC
VAR_IN_OUT
	AXIS : _AXIS_REF_REAL;
	DATA : ARRAY [1..L_MC1P_Constants.gc_Rec_MaxDataIndex] OF POINTER TO L_MC1P_MappedElement;
	DRIVESPECIFIC : L_MC1P_DriveSpecific_Generic;
END_VAR
END_METHOD

METHOD TRANSMITPARAMETERCALC
VAR_IN_OUT
	AXIS : _AXIS_REF_REAL;
	DATA : ARRAY [1..L_MC1P_Constants.gc_Trans_MaxDataIndex] OF POINTER TO L_MC1P_MappedElement;
	DRIVESPECIFIC : L_MC1P_DriveSpecific_Generic;
END_VAR
END_METHOD

(* ---- L_MC1P_ILMDATA.itf ---- *)
INTERFACE L_MC1P_ILMDATA
END_INTERFACE

METHOD ABORT : UDINT
END_METHOD

METHOD EXECUTE : UDINT
END_METHOD

(* ---- L_MC1P_IMANAGEMENTFUNCTION.itf ---- *)
INTERFACE L_MC1P_IMANAGEMENTFUNCTION
END_INTERFACE

METHOD COMPAREAXISNAME : BOOL
VAR_IN_OUT
	SAXISNAME : STRING;
END_VAR
END_METHOD

METHOD GETAXIS : POINTER TO AXIS_REF
END_METHOD

(* ---- L_MC1P_IMANIPULATEACTVALUES.itf ---- *)
INTERFACE L_MC1P_IMANIPULATEACTVALUES
END_INTERFACE

METHOD MANIPULATEACTVALUES
VAR_IN_OUT
	AXIS : AXIS_REF;
END_VAR
END_METHOD

(* ---- L_MC1P_IMANIPULATIONINTERFACE.itf ---- *)
INTERFACE L_MC1P_IMANIPULATIONINTERFACE
END_INTERFACE

METHOD CALCVALUES
VAR_INPUT
	XENABLE : BOOL;
	XRESET : BOOL;
	LRSETPOS : LREAL;
	LRSETVEL : LREAL;
	LRSETACC : LREAL;
	LRSETTORQUE : LREAL;
	XLOADPOSOFFSET : BOOL;
	LRPOSOFFSET : LREAL;
END_VAR
VAR_OUTPUT
	XACTIVE : BOOL;
	XERROR : BOOL;
	EERRORID : L_IE1P.L_IE1P_Error;
	LRSETPOSOUT : LREAL;
	LRSETVELOUT : LREAL;
	LRSETACCOUT : LREAL;
	LRSETTORQUEOUT : LREAL;
END_VAR
VAR_IN_OUT
	AXIS : Axis_REf;
END_VAR
END_METHOD

(* ---- L_MC1P_IMECHANICSIMULATION.itf ---- *)
INTERFACE L_MC1P_IMECHANICSIMULATION
END_INTERFACE

METHOD CALLMECHANICSIMULATION : BOOL
VAR_INPUT
	XBRAKERELEASED : BOOL;
	LRACTTORQUE : LREAL;
	LRTASKCYCLESYSSIM : LREAL;
	LRINVTASKCYCLESYSSIM : LREAL;
END_VAR
VAR_OUTPUT
	LRACTPOS : LREAL;
	LRACTVEL : LREAL;
END_VAR
END_METHOD

METHOD SCALEPARAMETER
END_METHOD

METHOD SETSTARTPOSITION : BOOL
VAR_INPUT
	LRPOS : LREAL;
END_VAR
END_METHOD

(* ---- L_MC1P_IMOLACCESS.itf ---- *)
INTERFACE L_MC1P_IMOLACCESS
END_INTERFACE

METHOD SETMOLSTATES
VAR_INPUT
	WSETMOLSTATE : WORD := 0;
	WSETMOLMODE : WORD := 0;
END_VAR
END_METHOD

(* ---- L_MC1P_IPARA.itf ---- *)
INTERFACE L_MC1P_IPARA
END_INTERFACE

METHOD HLP_GETPARAMETERPROPERTIES : BOOL
VAR_INPUT
	PAXISREF : POINTER TO AXIS_REF;
	DIPARAMETER : DINT;
	XALLOWINVISIBLE : BOOL;
END_VAR
VAR_OUTPUT
	PPARAMADDR : POINTER TO BYTE;
	EORDINALTYPE : L_MC1P_OrdinalType;
	XREADWRITE : BOOL;
	LRUNITFACTOR : LREAL;
	LRDEFAULTVALUE : LREAL;
	WVALUERANGES : WORD;
	PVALUERANGES : POINTER TO L_MC1P_MinMaxValue;
END_VAR
END_METHOD

METHOD HLP_READBOOLPARAMETER : BOOL
VAR_INPUT
	PINPUTDATA : POINTER TO BYTE;
	PARAMETER : DINT;
	PXVALUE : POINTER TO BOOL;
	XALLOWINVISIBLE : BOOL;
END_VAR
END_METHOD

METHOD HLP_READPARAMETER : BOOL
VAR_INPUT
	PINPUTDATA : POINTER TO BYTE;
	PARAMETER : DINT;
	PLRVALUE : POINTER TO LREAL;
	XALLOWINVISIBLE : BOOL;
END_VAR
END_METHOD

METHOD HLP_WRITEBOOLPARAMETER : BOOL
VAR_INPUT
	PINPUTDATA : POINTER TO BYTE;
	PARAMETER : DINT;
	PXVALUE : POINTER TO BOOL;
	XALLOWINVISIBLE : BOOL;
END_VAR
VAR_OUTPUT
	WERRORID : WORD;
END_VAR
END_METHOD

METHOD HLP_WRITEPARAMETER : BOOL
VAR_INPUT
	PINPUTDATA : POINTER TO BYTE;
	PARAMETER : DINT;
	PLRVALUE : POINTER TO LREAL;
	XALLOWINVISIBLE : BOOL;
END_VAR
VAR_OUTPUT
	WERRORID : WORD;
END_VAR
END_METHOD

(* ---- L_MC1P_IPLIACCESS.itf ---- *)
INTERFACE L_MC1P_IPLIACCESS
END_INTERFACE

METHOD SETPPISTATES
VAR_INPUT
	WSETPPISTATE : WORD := 0;
	WSETPPIMODE : WORD := 0;
END_VAR
END_METHOD

(* ---- L_MC1P_IPOSPROFILECALCULATION.itf ---- *)
INTERFACE L_MC1P_IPOSPROFILECALCULATION
END_INTERFACE

METHOD CALCPROFILEDATA
VAR_INPUT
	PPOSPROFILERDATA : POINTER TO L_MC1P_PosProfiler;
	LRSTARTACC : LREAL;
	LRSTARTVEL : LREAL;
	LRSTARTPOS : LREAL;
	XVELMODE : BOOL;
END_VAR
VAR_OUTPUT
	XERROR : BOOL;
	DWSTATE : DWORD;
	DWPROFILETYPE : DWORD;
END_VAR
VAR_IN_OUT
	SCPROFILEDATA : L_MC1P_ProfileData;
	SCPROFILEPARAMETER : L_MC1P_ProfileParameter;
END_VAR
END_METHOD

METHOD PROFILEINTERPOLATOR : BOOL
VAR_INPUT
	PPOSPROFILERDATA : POINTER TO L_MC1P_PosProfiler;
	LREVALTIME : LREAL;
END_VAR
VAR_OUTPUT
	DWSTATE : DWORD;
	LRSETPOS : LREAL;
	LRSETVEL : LREAL;
	LRSETACC : LREAL;
END_VAR
VAR_IN_OUT
	SCPROFILEDATA : L_MC1P_ProfileData;
END_VAR
END_METHOD

METHOD STRETCHPROFILE
VAR_INPUT
	PPOSPROFILERDATA : POINTER TO L_MC1P_PosProfiler;
	LRTIMEBASE : LREAL;
END_VAR
VAR_IN_OUT
	SCPROFILEDATA : L_MC1P_ProfileData;
END_VAR
END_METHOD

(* ---- L_MC1P_IPOSPROFILERACTIVE.itf ---- *)
INTERFACE L_MC1P_IPOSPROFILERACTIVE
END_INTERFACE

(* ---- L_MC1P_IPOSSIGNALPROCESSING.itf ---- *)
INTERFACE L_MC1P_IPOSSIGNALPROCESSING
END_INTERFACE

METHOD CALCULATE : DINT
VAR_INPUT
	DIACTPOS : DINT;
	DWSAMPLETIME : DWORD;
	DWACTTIME : DWORD;
END_VAR
VAR_OUTPUT
	DIPOSOUT : DINT;
	XVELVALID : BOOL;
	DIVELOUT : DINT;
END_VAR
VAR_IN_OUT
	AXIS : _AXIS_REF_REAL;
END_VAR
END_METHOD

(* ---- L_MC1P_IRETAINFUNCTION.itf ---- *)
INTERFACE L_MC1P_IRETAINFUNCTION
END_INTERFACE

METHOD GETINITIALDATA : BOOL
VAR_INPUT
	PDATA : POINTER TO DWORD;
	INFO : DWORD;
END_VAR
END_METHOD

METHOD SETERRORINFO
VAR_INPUT
	WSTATE : WORD;
END_VAR
END_METHOD

METHOD SETINITIALDATA : BOOL
VAR_INPUT
	PDATA : POINTER TO DWORD;
END_VAR
END_METHOD

METHOD STOREDATA
VAR_INPUT
	PDATA : POINTER TO DWORD;
END_VAR
END_METHOD

(* ---- L_MC1P_IRETAINHANDLING.itf ---- *)
INTERFACE L_MC1P_IRETAINHANDLING
END_INTERFACE

METHOD GETINITIALRETAINDATA : POINTER TO L_MC1P_uRetainData
VAR_INPUT
	XNEWEST : BOOL;
END_VAR
END_METHOD

METHOD GETRETAINSTATE : WORD
VAR_OUTPUT
	WSTATERETAINERROR : WORD;
END_VAR
END_METHOD

METHOD REGISTERONRETAINDATAHANDLER
VAR_INPUT
	AXISGUID : L_MC1P_AxisGUID;
END_VAR
END_METHOD

METHOD RESET
END_METHOD

METHOD SETCONNECTEDGUID : BOOL
VAR_INPUT
	GUID : L_MC1P_AxisGUID;
END_VAR
END_METHOD

(* ---- L_MC1P_ISETVALUEMANIPULATIONINTERFACE.itf ---- *)
INTERFACE L_MC1P_ISETVALUEMANIPULATIONINTERFACE
END_INTERFACE

(* ---- L_MC1P_ITPSOURCEAXIS.itf ---- *)
INTERFACE L_MC1P_ITPSOURCEAXIS
END_INTERFACE

METHOD GETPOINTERTOTPAXIS : POINTER TO _AXIS_REF_REAL
END_METHOD

(* ---- GETBOOLEANPROPERTY.pou ---- *)
FUNCTION GETBOOLEANPROPERTY : BOOL
VAR_INPUT
	STKEY : WSTRING;
END_VAR
END_FUNCTION

(* ---- GETCOMPANY.pou ---- *)
FUNCTION GETCOMPANY : WSTRING
END_FUNCTION

(* ---- GETNUMBERPROPERTY.pou ---- *)
FUNCTION GETNUMBERPROPERTY : DINT
VAR_INPUT
	STKEY : WSTRING;
END_VAR
END_FUNCTION

(* ---- GETTEXTPROPERTY.pou ---- *)
FUNCTION GETTEXTPROPERTY : WSTRING
VAR_INPUT
	STKEY : WSTRING;
END_VAR
END_FUNCTION

(* ---- GETTEXTPROPERTY2.pou ---- *)
FUNCTION GETTEXTPROPERTY2 : POINTER TO WSTRING
VAR_INPUT
	STKEY : WSTRING;
END_VAR
END_FUNCTION

(* ---- GETTITLE.pou ---- *)
FUNCTION GETTITLE : WSTRING
END_FUNCTION

(* ---- GETVERSION.pou ---- *)
FUNCTION GETVERSION : VERSION
END_FUNCTION

(* ---- GETVERSIONPROPERTY.pou ---- *)
FUNCTION GETVERSIONPROPERTY : VERSION
VAR_INPUT
	STKEY : WSTRING;
END_VAR
END_FUNCTION

(* ---- L_MC1P_CHECKFORSENSORLESMODEIXXX.pou ---- *)
FUNCTION L_MC1P_CHECKFORSENSORLESMODEIXXX : BOOL
VAR_INPUT
	WMCTRLMODE : WORD;
END_VAR
END_FUNCTION

(* ---- L_MC1P_CODENUMBERTOPARAMETER.pou ---- *)
FUNCTION L_MC1P_CODENUMBERTOPARAMETER : DINT
VAR_INPUT
	DWCODENUMBER : DWORD;
	USISUBINDEX : USINT;
	UIBYTELENGTH : UINT;
END_VAR
END_FUNCTION

(* ---- L_MC1P_CODENUMBERTOPARAMETER2.pou ---- *)
FUNCTION L_MC1P_CODENUMBERTOPARAMETER2 : DINT
VAR_INPUT
	DWCODENUMBER : DWORD;
	USISUBINDEX : USINT;
	UIBYTELENGTH : UINT;
	XUNSIGNED : BOOL := FALSE;
END_VAR
END_FUNCTION

(* ---- L_MC1P_CONVERTPOSTOMODULOPOS.pou ---- *)
FUNCTION L_MC1P_CONVERTPOSTOMODULOPOS : LREAL
VAR_INPUT
	LRPOS : LREAL;
	LRPERIOD : LREAL;
END_VAR
END_FUNCTION

(* ---- L_MC1P_CONVERTPOSTOMODULOPOSEXTENDED.pou ---- *)
FUNCTION L_MC1P_CONVERTPOSTOMODULOPOSEXTENDED : LREAL
VAR_INPUT
	LRPOS : LREAL;
	LRPERIOD : LREAL;
END_VAR
END_FUNCTION

(* ---- L_MC1P_CONVERTPOSTOMODULOPOSFMOD.pou ---- *)
FUNCTION L_MC1P_CONVERTPOSTOMODULOPOSFMOD : LREAL
VAR_INPUT
	LRPOS : LREAL;
	LRPERIOD : LREAL;
END_VAR
END_FUNCTION

(* ---- L_MC1P_DIV.pou ---- *)
FUNCTION L_MC1P_DIV : LREAL
VAR_INPUT
	A : LREAL;
	B : LREAL;
END_VAR
END_FUNCTION

(* ---- L_MC1P_FINDDRIVECONNECTORFROMENCODER.pou ---- *)
FUNCTION L_MC1P_FINDDRIVECONNECTORFROMENCODER : POINTER TO IoConfigConnector
VAR_INPUT
	PCONNECTOR : POINTER TO IoConfigConnector;
END_VAR
END_FUNCTION

(* ---- L_MC1P_FINDOWNSLICEPOSITIONS131.pou ---- *)
FUNCTION L_MC1P_FINDOWNSLICEPOSITIONS131 : BOOL
VAR_INPUT
	M_PCONNECTOR : POINTER TO IoConfigConnector;
END_VAR
VAR_OUTPUT
	WSLICEPOSITION : WORD;
END_VAR
END_FUNCTION

(* ---- L_MC1P_FINDPDODATAINCONNECTOR.pou ---- *)
FUNCTION L_MC1P_FINDPDODATAINCONNECTOR : POINTER TO BYTE
VAR_INPUT
	PCONNECTOR : POINTER TO IoConfigConnector;
	UIINDEX : WORD;
	USISUBINDEX : USINT;
	XWRITEACCESS : BOOL;
END_VAR
VAR_OUTPUT
	USISIZE : USINT;
END_VAR
END_FUNCTION

(* ---- L_MC1P_GENTIMESTAMPSIMU.pou ---- *)
FUNCTION L_MC1P_GENTIMESTAMPSIMU : WORD
VAR_IN_OUT
	AXIS : AXIS_REF;
END_VAR
END_FUNCTION

(* ---- L_MC1P_GETDIGINPUTSFROMDRIVE.pou ---- *)
FUNCTION L_MC1P_GETDIGINPUTSFROMDRIVE : DWORD
VAR_IN_OUT
	AXIS : AXIS_REF;
END_VAR
END_FUNCTION

(* ---- L_MC1P_GETINSTANCENAME.pou ---- *)
FUNCTION L_MC1P_GETINSTANCENAME : STRING(L_MC1P_Constants.gc_wInstanceNchar)
VAR_INPUT
	SSTR : STRING(L_MC1P_Constants.gc_wInstanceNchar);
END_VAR
END_FUNCTION

(* ---- L_MC1P_GETIOMGRCONFIGCONNECTORLIST.pou ---- *)
FUNCTION L_MC1P_GETIOMGRCONFIGCONNECTORLIST : SysTypes.RTS_IEC_RESULT
VAR_INPUT
	PPCONNECTORLIST : POINTER TO POINTER TO IoConfigConnector;
	PNCOUNT : POINTER TO DINT;
END_VAR
END_FUNCTION

(* ---- L_MC1P_GETIOMGRCONFIGFINDCONNETOR.pou ---- *)
FUNCTION L_MC1P_GETIOMGRCONFIGFINDCONNETOR : POINTER TO IoConfigConnector
VAR_INPUT
	PCONNECTOR : POINTER TO IoConfigConnector;
END_VAR
VAR_OUTPUT
	NCOUNT : DINT := 0;
END_VAR
END_FUNCTION

(* ---- L_MC1P_GETIOMGRCONFIGFIRSTCHILD.pou ---- *)
FUNCTION L_MC1P_GETIOMGRCONFIGFIRSTCHILD : POINTER TO IoConfigConnector
VAR_INPUT
	PIOCONNECTORLIST : POINTER TO IoConfigConnector;
	PNCOUNT : POINTER TO DINT;
	PFATHER : POINTER TO IoConfigConnector;
END_VAR
END_FUNCTION

(* ---- L_MC1P_GETIOMGRCONFIGNEXTCHILD.pou ---- *)
FUNCTION L_MC1P_GETIOMGRCONFIGNEXTCHILD : POINTER TO IoConfigConnector
VAR_INPUT
	PIOCONNECTORLIST : POINTER TO IoConfigConnector;
	PNCOUNT : POINTER TO DINT;
	PFATHER : POINTER TO IoConfigConnector;
END_VAR
END_FUNCTION

(* ---- L_MC1P_GETIOMGRCONFIGPARAMETER.pou ---- *)
FUNCTION L_MC1P_GETIOMGRCONFIGPARAMETER : POINTER TO IoConfigParameter
VAR_INPUT
	PCONNECTOR : POINTER TO IoConfigConnector;
	DWPARAMETERID : DWORD;
END_VAR
END_FUNCTION

(* ---- L_MC1P_GETIOMGRCONFIGPARAMETERVALUEBYTE.pou ---- *)
FUNCTION L_MC1P_GETIOMGRCONFIGPARAMETERVALUEBYTE : BYTE
VAR_INPUT
	PPARAMETER : POINTER TO IoConfigParameter;
	PRESULT : POINTER TO UDINT;
END_VAR
END_FUNCTION

(* ---- L_MC1P_GETIOMGRCONFIGPARAMETERVALUEDWORD.pou ---- *)
FUNCTION L_MC1P_GETIOMGRCONFIGPARAMETERVALUEDWORD : DWORD
VAR_INPUT
	PPARAMETER : POINTER TO IoConfigParameter;
	PRESULT : POINTER TO UDINT;
END_VAR
END_FUNCTION

(* ---- L_MC1P_GETIOMGRCONFIGPARAMETERVALUEWORD.pou ---- *)
FUNCTION L_MC1P_GETIOMGRCONFIGPARAMETERVALUEWORD : WORD
VAR_INPUT
	PPARAMETER : POINTER TO IoConfigParameter;
	PRESULT : POINTER TO UDINT;
END_VAR
END_FUNCTION

(* ---- L_MC1P_GETRATEDTORQUEAXIS.pou ---- *)
FUNCTION L_MC1P_GETRATEDTORQUEAXIS : LREAL
VAR_IN_OUT
	AXIS : AXIS_REF;
END_VAR
END_FUNCTION

(* ---- L_MC1P_GETRATEDVELOCITYAXIS.pou ---- *)
FUNCTION L_MC1P_GETRATEDVELOCITYAXIS : LREAL
VAR_IN_OUT
	AXIS : AXIS_REF;
END_VAR
END_FUNCTION

(* ---- L_MC1P_GETTASKCYCLE.pou ---- *)
FUNCTION L_MC1P_GETTASKCYCLE : LREAL
END_FUNCTION

(* ---- L_MC1P_HLPABSDINT.pou ---- *)
FUNCTION L_MC1P_HLPABSDINT : DINT
VAR_INPUT
	DIVAR : DINT;
END_VAR
END_FUNCTION

(* ---- L_MC1P_HLPCALCPOLY5THORDERSCALED.pou ---- *)
FUNCTION L_MC1P_HLPCALCPOLY5THORDERSCALED : LREAL
VAR_OUTPUT
	LRYPOSSCALED : LREAL;
END_VAR
VAR_IN_OUT
	LRXPOSSCALED : LREAL;
	ALRKOEF : ARRAY [0..5] OF LREAL;
END_VAR
END_FUNCTION

(* ---- L_MC1P_HLPCHECKDIRECTION.pou ---- *)
FUNCTION L_MC1P_HLPCHECKDIRECTION : INT
VAR_IN_OUT
	LRPOSFIFOX : ARRAY [1..20] OF LREAL;
	LRLEN : LREAL;
END_VAR
END_FUNCTION

(* ---- L_MC1P_HLPDELTAVELTIMEEXTENDED.pou ---- *)
FUNCTION L_MC1P_HLPDELTAVELTIMEEXTENDED : BOOL
VAR_INPUT
	LRVELSTART : LREAL;
	LRACCSTART : LREAL;
	LRMAXACC : LREAL;
	LRMAXJERK : LREAL;
END_VAR
VAR_OUTPUT
	LRTIME : LREAL;
	LRDIST : LREAL;
END_VAR
END_FUNCTION

(* ---- L_MC1P_HLPFITCYCLELIM.pou ---- *)
FUNCTION L_MC1P_HLPFITCYCLELIM : BOOL
VAR_INPUT
	PLRPOS : POINTER TO LREAL;
	LRLEN : LREAL;
END_VAR
END_FUNCTION

(* ---- L_MC1P_HLPGEARRES.pou ---- *)
FUNCTION L_MC1P_HLPGEARRES : LREAL
VAR_INPUT
	LRINPUT : LREAL;
	LRNUM : LREAL;
	LRDEN : LREAL;
END_VAR
END_FUNCTION

(* ---- L_MC1P_HLPMODULOADD.pou ---- *)
FUNCTION L_MC1P_HLPMODULOADD : LREAL
VAR_INPUT
	LRINPUT : LREAL;
	LROFFSET : LREAL;
	LRLENGHT : LREAL;
END_VAR
END_FUNCTION

(* ---- L_MC1P_HLPMODULODIFF.pou ---- *)
FUNCTION L_MC1P_HLPMODULODIFF : LREAL
VAR_INPUT
	LRDIFF : LREAL;
	LRLEN : LREAL;
END_VAR
END_FUNCTION

(* ---- L_MC1P_HLPMODULOOFFSET.pou ---- *)
FUNCTION L_MC1P_HLPMODULOOFFSET : LREAL
VAR_INPUT
	LROFFSET : LREAL;
	LRLENGTH : LREAL;
	PLROFFSETBASE : POINTER TO LREAL;
END_VAR
END_FUNCTION

(* ---- L_MC1P_HLPMODULOSUB.pou ---- *)
FUNCTION L_MC1P_HLPMODULOSUB : LREAL
VAR_INPUT
	LRDIFF : LREAL;
	LRLEN : LREAL;
END_VAR
END_FUNCTION

(* ---- L_MC1P_HLPMODULOZEROPOS.pou ---- *)
FUNCTION L_MC1P_HLPMODULOZEROPOS : BOOL
VAR_INPUT
	PLRPOS : POINTER TO LREAL;
	LRLENINT : LREAL;
END_VAR
END_FUNCTION

(* ---- L_MC1P_HLPPOLY4RG.pou ---- *)
FUNCTION L_MC1P_HLPPOLY4RG : LREAL
VAR_INPUT
	LRX : LREAL;
END_VAR
END_FUNCTION

(* ---- L_MC1P_HLPPT1FILT.pou ---- *)
FUNCTION L_MC1P_HLPPT1FILT : LREAL
VAR_INPUT
	LRVALUE : LREAL;
	LRINPUT : LREAL;
	LRNEW_N : LREAL;
END_VAR
END_FUNCTION

(* ---- L_MC1P_HLPSIGNNE.pou ---- *)
FUNCTION L_MC1P_HLPSIGNNE : BOOL
VAR_INPUT
	A : LREAL;
	B : LREAL;
END_VAR
END_FUNCTION

(* ---- L_MC1P_INDEXTOPARAMETER.pou ---- *)
FUNCTION L_MC1P_INDEXTOPARAMETER : DINT
VAR_INPUT
	UIINDEX : UINT;
	USISUBINDEX : USINT;
	UIBYTELENGTH : UINT := 4;
END_VAR
END_FUNCTION

(* ---- L_MC1P_INDEXTOPARAMETER2.pou ---- *)
FUNCTION L_MC1P_INDEXTOPARAMETER2 : DINT
VAR_INPUT
	UIINDEX : UINT;
	USISUBINDEX : USINT;
	UIBYTELENGTH : UINT := 4;
	XUNSIGNED : BOOL := FALSE;
END_VAR
END_FUNCTION

(* ---- L_MC1P_LMDATAMANAGERINSERTDATA.pou ---- *)
FUNCTION L_MC1P_LMDATAMANAGERINSERTDATA : BOOL
VAR_INPUT
	ITFLMDATA : L_MC1P_ILMData;
END_VAR
END_FUNCTION

(* ---- L_MC1P_LREAL_TO_DINT.pou ---- *)
FUNCTION L_MC1P_LREAL_TO_DINT : DINT
VAR_INPUT
	LRVALUE : LREAL;
END_VAR
END_FUNCTION

(* ---- L_MC1P_LREAL_TO_DINT_TO_DWORD.pou ---- *)
FUNCTION L_MC1P_LREAL_TO_DINT_TO_DWORD : DWORD
VAR_INPUT
	LRVALUE : LREAL;
END_VAR
END_FUNCTION

(* ---- L_MC1P_LREAL_TO_DWORD.pou ---- *)
FUNCTION L_MC1P_LREAL_TO_DWORD : DWORD
VAR_INPUT
	LRVALUE : LREAL;
END_VAR
END_FUNCTION

(* ---- L_MC1P_LREAL_TO_INT.pou ---- *)
FUNCTION L_MC1P_LREAL_TO_INT : INT
VAR_INPUT
	LRVALUE : LREAL;
END_VAR
END_FUNCTION

(* ---- L_MC1P_LREAL_TO_INT_TO_WORD.pou ---- *)
FUNCTION L_MC1P_LREAL_TO_INT_TO_WORD : WORD
VAR_INPUT
	LRVALUE : LREAL;
END_VAR
END_FUNCTION

(* ---- L_MC1P_LREAL_TO_WORD.pou ---- *)
FUNCTION L_MC1P_LREAL_TO_WORD : WORD
VAR_INPUT
	LRVALUE : LREAL;
END_VAR
END_FUNCTION

(* ---- L_MC1P_LREQ.pou ---- *)
FUNCTION L_MC1P_LREQ : BOOL
VAR_INPUT
	LRVALUE : LREAL;
	LRTARGET : LREAL;
END_VAR
END_FUNCTION

(* ---- L_MC1P_LRGE.pou ---- *)
FUNCTION L_MC1P_LRGE : BOOL
VAR_INPUT
	LRVALUE : LREAL;
	LRTARGET : LREAL;
END_VAR
END_FUNCTION

(* ---- L_MC1P_LRGT.pou ---- *)
FUNCTION L_MC1P_LRGT : BOOL
VAR_INPUT
	LRVALUE : LREAL;
	LRTARGET : LREAL;
END_VAR
END_FUNCTION

(* ---- L_MC1P_LRLE.pou ---- *)
FUNCTION L_MC1P_LRLE : BOOL
VAR_INPUT
	LRVALUE : LREAL;
	LRTARGET : LREAL;
END_VAR
END_FUNCTION

(* ---- L_MC1P_LRLT.pou ---- *)
FUNCTION L_MC1P_LRLT : BOOL
VAR_INPUT
	LRVALUE : LREAL;
	LRTARGET : LREAL;
END_VAR
END_FUNCTION

(* ---- L_MC1P_LRNE.pou ---- *)
FUNCTION L_MC1P_LRNE : BOOL
VAR_INPUT
	LRVALUE : LREAL;
	LRTARGET : LREAL;
END_VAR
END_FUNCTION

(* ---- L_MC1P_MODULOCYCLE.pou ---- *)
FUNCTION L_MC1P_MODULOCYCLE : LREAL
VAR_INPUT
	LRPOSIN : LREAL;
	LRPOSITIONPERIOD : LREAL;
END_VAR
END_FUNCTION

(* ---- L_MC1P_POS_DINT_TO_LINT.pou ---- *)
FUNCTION L_MC1P_POS_DINT_TO_LINT : LINT
VAR_INPUT
	DIPOS : DINT;
	DIPOSOLD : DINT;
END_VAR
VAR_IN_OUT
	UPOS : L_MC1P_PosLINT;
END_VAR
END_FUNCTION

(* ---- L_MC1P_POSDIFFTOSPEEDINCIXXX.pou ---- *)
FUNCTION L_MC1P_POSDIFFTOSPEEDINCIXXX : DINT
VAR_INPUT
	DIPOSDIFF : DINT := 0;
	DWFACTOR : DWORD := 1000;
	DWINKPERREV : DWORD := 65536;
END_VAR
END_FUNCTION

(* ---- L_MC1P_SPEEDTOPOSDIFFINCIXXX.pou ---- *)
FUNCTION L_MC1P_SPEEDTOPOSDIFFINCIXXX : DINT
VAR_INPUT
	DISPEED : DINT := 0;
	DWFACTOR : DWORD := 1000;
	DWINKPERREV : DWORD := 65536;
END_VAR
VAR_IN_OUT
	DIRES : DINT;
END_VAR
END_FUNCTION

(* ---- L_MC1P_STVARIABLENAME_TO_DWORD.pou ---- *)
FUNCTION L_MC1P_STVARIABLENAME_TO_DWORD : BOOL
VAR_INPUT
	STVARIABLENAME : STRING;
END_VAR
VAR_OUTPUT
	DWOUT : DWORD;
END_VAR
END_FUNCTION

(* ---- L_MC1P_STVARIABLENAME_TO_INT.pou ---- *)
FUNCTION L_MC1P_STVARIABLENAME_TO_INT : BOOL
VAR_INPUT
	STVARIABLENAME : STRING;
END_VAR
VAR_OUTPUT
	IOUT : INT;
END_VAR
END_FUNCTION

(* ---- L_MC1P_STVARIABLENAME_TO_LREAL.pou ---- *)
FUNCTION L_MC1P_STVARIABLENAME_TO_LREAL : BOOL
VAR_INPUT
	STVARIABLENAME : STRING(255);
END_VAR
VAR_OUTPUT
	LROUT : LREAL;
END_VAR
END_FUNCTION

(* ---- L_MC1P_STVARIABLENAME_TO_REAL.pou ---- *)
FUNCTION L_MC1P_STVARIABLENAME_TO_REAL : BOOL
VAR_INPUT
	STVARIABLENAME : STRING;
END_VAR
VAR_OUTPUT
	ROUT : REAL;
END_VAR
END_FUNCTION

(* ---- L_MC1P_STVARIABLENAME_TO_WORD.pou ---- *)
FUNCTION L_MC1P_STVARIABLENAME_TO_WORD : BOOL
VAR_INPUT
	STVARIABLENAME : STRING;
END_VAR
VAR_OUTPUT
	WOUT : WORD;
END_VAR
END_FUNCTION

(* ---- L_MC1P_TRUNC_LINT.pou ---- *)
FUNCTION L_MC1P_TRUNC_LINT : LINT
VAR_INPUT
	LRIN : LREAL;
END_VAR
END_FUNCTION

(* ---- L_MC1P_USEHOMINGPOSITIONFROMAXISREF.pou ---- *)
FUNCTION L_MC1P_USEHOMINGPOSITIONFROMAXISREF : BOOL
VAR_INPUT
	XACTIVATE : BOOL;
END_VAR
VAR_IN_OUT
	AXIS : AXIS_REF;
END_VAR
END_FUNCTION

(* ---- L_MC1P_USEMANUALPARAMETERFROMAXISREF.pou ---- *)
FUNCTION L_MC1P_USEMANUALPARAMETERFROMAXISREF : BOOL
VAR_INPUT
	XACTIVATE : BOOL;
END_VAR
VAR_IN_OUT
	AXIS : AXIS_REF;
END_VAR
END_FUNCTION

(* ---- _AXIS_REF_9400HL.pou ---- *)
FUNCTION_BLOCK _AXIS_REF_9400HL EXTENDS _AXIS_REF_COM
VAR
	AXISEXTENSION : L_MC1P_AxisExtension_9400HL;
	MOTIONUTILS : L_MC1P_MotionUtils_9400HL;
	RETAINMANAGEMENT : L_MC1P_MotionUtilsRetainHandling;
END_VAR
END_FUNCTION_BLOCK

METHOD FB_INIT : BOOL
VAR_INPUT
	BINITRETAINS : BOOL;
	BINCOPYCODE : BOOL;
END_VAR
END_METHOD

(* ---- _AXIS_REF_9400HL_CAN.pou ---- *)
FUNCTION_BLOCK _AXIS_REF_9400HL_CAN EXTENDS _AXIS_REF_COM
VAR
	AXISEXTENSION : L_MC1P_AxisExtension_9400HL_CAN;
	MOTIONUTILS : L_MC1P_MotionUtils_9400HL_CAN;
	RETAINMANAGEMENT : L_MC1P_MotionUtilsRetainHandling;
END_VAR
END_FUNCTION_BLOCK

METHOD FB_INIT : BOOL
VAR_INPUT
	BINITRETAINS : BOOL;
	BINCOPYCODE : BOOL;
END_VAR
END_METHOD

(* ---- _AXIS_REF_COM.pou ---- *)
FUNCTION_BLOCK _AXIS_REF_COM EXTENDS _AXIS_REF_REAL
VAR
	WFATHERCONNECTORTYPE : WORD := L_MC1P_Constants.c_ConnectorTypeMotionAxisOld;
	WFATHERCONNECTORTYPE2 : WORD := L_MC1P_Constants.c_ConnectorTypeMotionAxis;
	HEVENTCOMMCYCLE : SysTypes.RTS_IEC_HANDLE := SysTypes.RTS_INVALID_HANDLE;
	HINTERFACECOMMCYCLE : SysTypes.RTS_IEC_HANDLE := SysTypes.RTS_INVALID_HANDLE;
	COMMCYCLECOUNT : DWORD;
	XCOMMERROR : BOOL;
	XCOMMWARNING : BOOL;
	WAITFORAXISDETECTION : BOOL;
END_VAR
END_FUNCTION_BLOCK

METHOD CONNECTASYNC : BOOL
END_METHOD

METHOD CALLSDODATAHANDLING
END_METHOD

METHOD CHECKCOMMUNCATION
END_METHOD

METHOD CHECKCOMMUNICATIONACYCLIC : BOOL
END_METHOD

METHOD GETMAPPEDDATA : POINTER TO BYTE
VAR_INPUT
	UIINDEX : WORD;
	USISUBINDEX : USINT;
	USISIZE : USINT;
	XWRITEACCESS : BOOL;
	PADDDATA : POINTER TO BYTE;
	PXWAITFORINITACCESS : POINTER TO BOOL;
END_VAR
VAR_OUTPUT
	EERRORID : L_IE1P_Error;
	XERROR : BOOL;
	USISIZEACT : USINT := 0;
END_VAR
END_METHOD

METHOD GETMAPPEDDATASUPPORT : BOOL
END_METHOD

METHOD HANDLESDOREADONCOMMERROR : BOOL
VAR_INPUT
	IDX : DWORD;
END_VAR
VAR_IN_OUT
	SDOREADDATA : L_DCO_SdoData;
END_VAR
END_METHOD

METHOD HANDLESDOWRITEONCOMMERROR : BOOL
VAR_INPUT
	IDX : DWORD;
END_VAR
VAR_IN_OUT
	SDOWRITEDATA : L_DCO_SdoData;
END_VAR
END_METHOD

METHOD CONFIGUREAXIS
END_METHOD

METHOD CONFIGUREAXIS2
END_METHOD

METHOD RESETAXISCONNECTOR
END_METHOD

METHOD UPDATEFATHERCONNECTOR
END_METHOD

METHOD SETAXISSIMULATION : BOOL
VAR_INPUT
	ITFAXISSIMULATION : L_MC1P_IAxisSimulationInterface;
END_VAR
END_METHOD

METHOD EVENTCALLBACK : UDINT
VAR_INPUT
	PEVENTPARAM : POINTER TO EventParam;
END_VAR
END_METHOD

METHOD REGISTEREVENT
END_METHOD

METHOD UNREGISTEREVENT
END_METHOD

METHOD GETIECADRESS
END_METHOD
